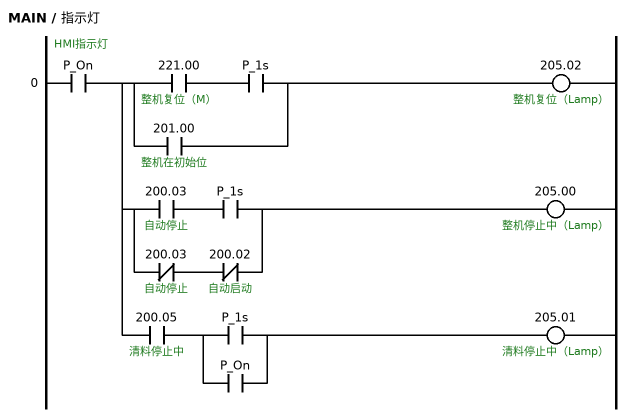
; [picture p336: MAIN / 指示灯, rungs 0-0]
; rung 0: HMI指示灯
LD P_On
OUT TR0
LD 221.00  ; 整机复位（M）
AND P_1s
OR 201.00  ; 整机在初始位
ANDLD
OUT 205.02  ; 整机复位（Lamp）
LD TR0
LD 200.03  ; 自动停止
AND P_1s
LDNOT 200.03  ; 自动停止
ANDNOT 200.02  ; 自动启动
ORLD
ANDLD
OUT 205.00  ; 整机停止中（Lamp）
LD TR0
AND 200.05  ; 清料停止中
LD P_1s
OR P_On
ANDLD
OUT 205.01  ; 清料停止中（Lamp）

### Section 外部输出

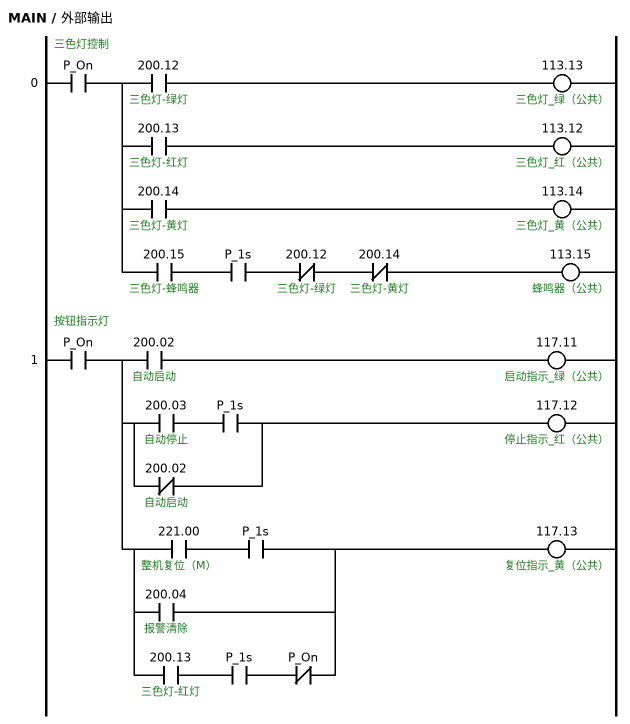
; rung 0: 三色灯控制
LD P_On
OUT TR0
AND 200.12  ; 三色灯-绿灯
OUT 113.13  ; 三色灯_绿（公共）
LD TR0
AND 200.13  ; 三色灯-红灯
OUT 113.12  ; 三色灯_红（公共）
LD TR0
AND 200.14  ; 三色灯-黄灯
OUT 113.14  ; 三色灯_黄（公共）
LD TR0
AND 200.15  ; 三色灯-蜂鸣器
AND P_1s
ANDNOT 200.12  ; 三色灯-绿灯
ANDNOT 200.14  ; 三色灯-黄灯
OUT 113.15  ; 蜂鸣器（公共）
; rung 1: 按钮指示灯
LD P_On
OUT TR0
AND 200.02  ; 自动启动
OUT 117.11  ; 启动指示_绿（公共）
LD TR0
LD 200.03  ; 自动停止
AND P_1s
ORNOT 200.02  ; 自动启动
ANDLD
OUT 117.12  ; 停止指示_红（公共）
LD TR0
LD 221.00  ; 整机复位（M）
AND P_1s
OR 200.04  ; 报警清除
LD 200.13  ; 三色灯-红灯
AND P_1s
ANDNOT P_On
ORLD
ANDLD
OUT 117.13  ; 复位指示_黄（公共）

### Section END
; rung 0
END(001)

## Program 电芯来料_RK_01 (cyclic task 1)

### Section Main

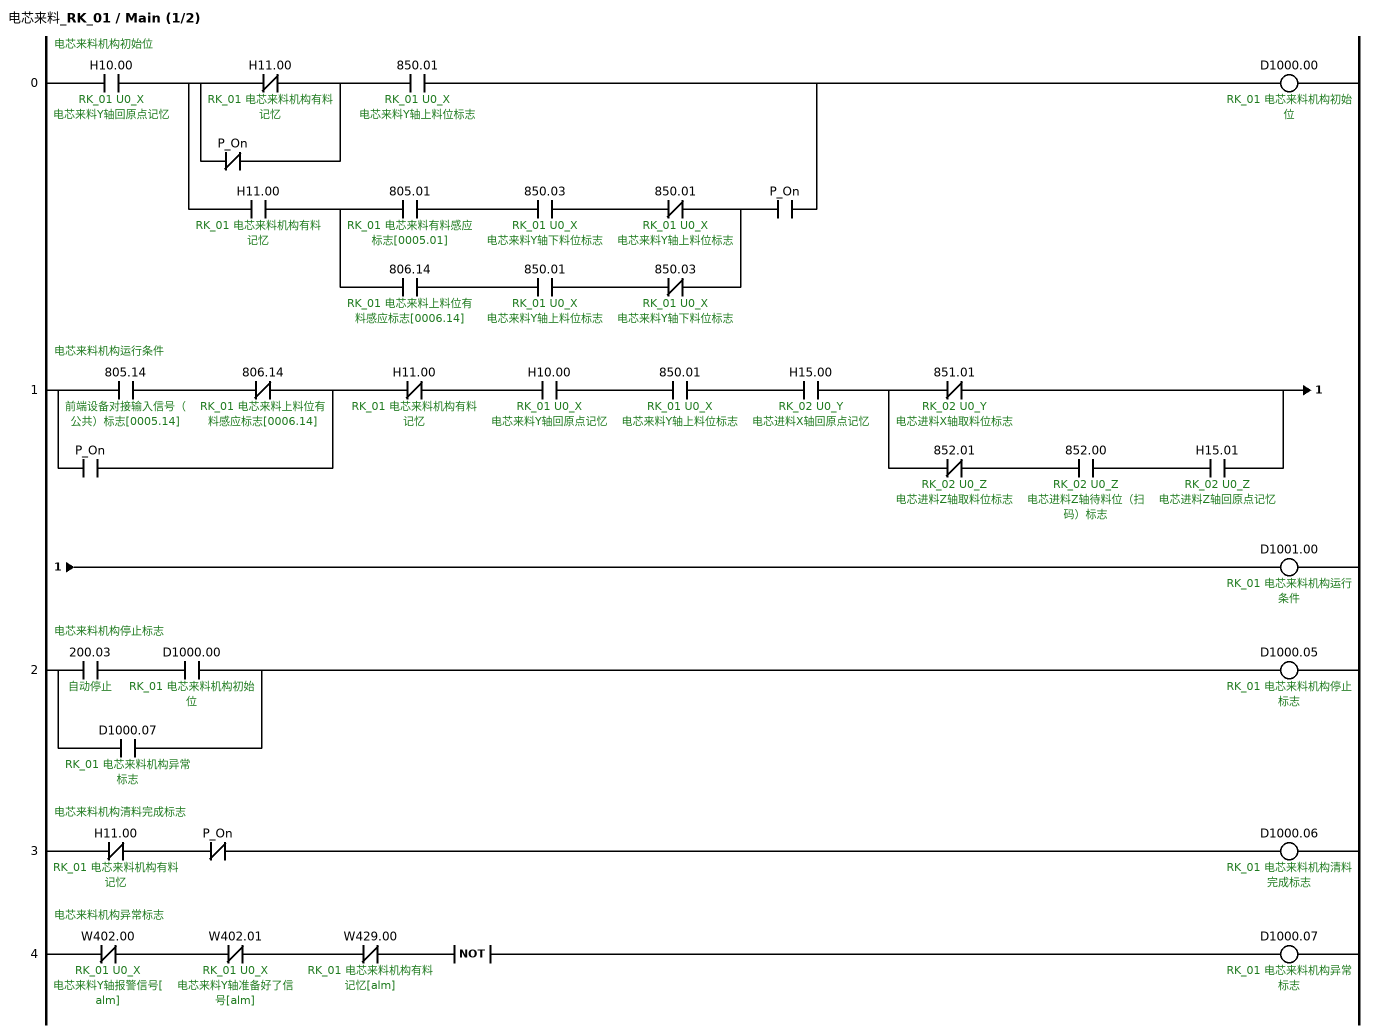
; rung 0: 电芯来料机构初始位
LD H10.00  ; RK_01 U0_X 电芯来料Y轴回原点记忆
LDNOT H11.00  ; RK_01 电芯来料机构有料记忆
ORNOT P_On
AND 850.01  ; RK_01 U0_X 电芯来料Y轴上料位标志
LD H11.00  ; RK_01 电芯来料机构有料记忆
LD 805.01  ; RK_01 电芯来料有料感应标志[0005.01]
AND 850.03  ; RK_01 U0_X 电芯来料Y轴下料位标志
ANDNOT 850.01  ; RK_01 U0_X 电芯来料Y轴上料位标志
LD 806.14  ; RK_01 电芯来料上料位有料感应标志[0006.14]
AND 850.01  ; RK_01 U0_X 电芯来料Y轴上料位标志
ANDNOT 850.03  ; RK_01 U0_X 电芯来料Y轴下料位标志
ORLD
ANDLD
AND P_On
ORLD
ANDLD
OUT D1000.00  ; RK_01 电芯来料机构初始位
; rung 1: 电芯来料机构运行条件
LD 805.14  ; 前端设备对接输入信号（公共）标志[0005.14]  // 前端设备放料中（放料中=1）！
ANDNOT 806.14  ; RK_01 电芯来料上料位有料感应标志[0006.14]
OR P_On
ANDNOT H11.00  ; RK_01 电芯来料机构有料记忆
AND H10.00  ; RK_01 U0_X 电芯来料Y轴回原点记忆
AND 850.01  ; RK_01 U0_X 电芯来料Y轴上料位标志
AND H15.00  ; RK_02 U0_Y 电芯进料X轴回原点记忆
LDNOT 851.01  ; RK_02 U0_Y 电芯进料X轴取料位标志
LDNOT 852.01  ; RK_02 U0_Z 电芯进料Z轴取料位标志
AND 852.00  ; RK_02 U0_Z 电芯进料Z轴待料位（扫码）标志
AND H15.01  ; RK_02 U0_Z 电芯进料Z轴回原点记忆
ORLD
ANDLD
OUT D1001.00  ; RK_01 电芯来料机构运行条件
; rung 2: 电芯来料机构停止标志
LD 200.03  ; 自动停止
AND D1000.00  ; RK_01 电芯来料机构初始位
OR D1000.07  ; RK_01 电芯来料机构异常标志
OUT D1000.05  ; RK_01 电芯来料机构停止标志
; rung 3: 电芯来料机构清料完成标志
LDNOT H11.00  ; RK_01 电芯来料机构有料记忆
ANDNOT P_On  // 上料位非扫码完成料，清料时无需考虑！！
OUT D1000.06  ; RK_01 电芯来料机构清料完成标志
; rung 4: 电芯来料机构异常标志
LDNOT W402.00  ; RK_01 U0_X 电芯来料Y轴报警信号[alm]
ANDNOT W402.01  ; RK_01 U0_X 电芯来料Y轴准备好了信号[alm]
ANDNOT W429.00  ; RK_01 电芯来料机构有料记忆[alm]
NOT(520)
OUT D1000.07  ; RK_01 电芯来料机构异常标志

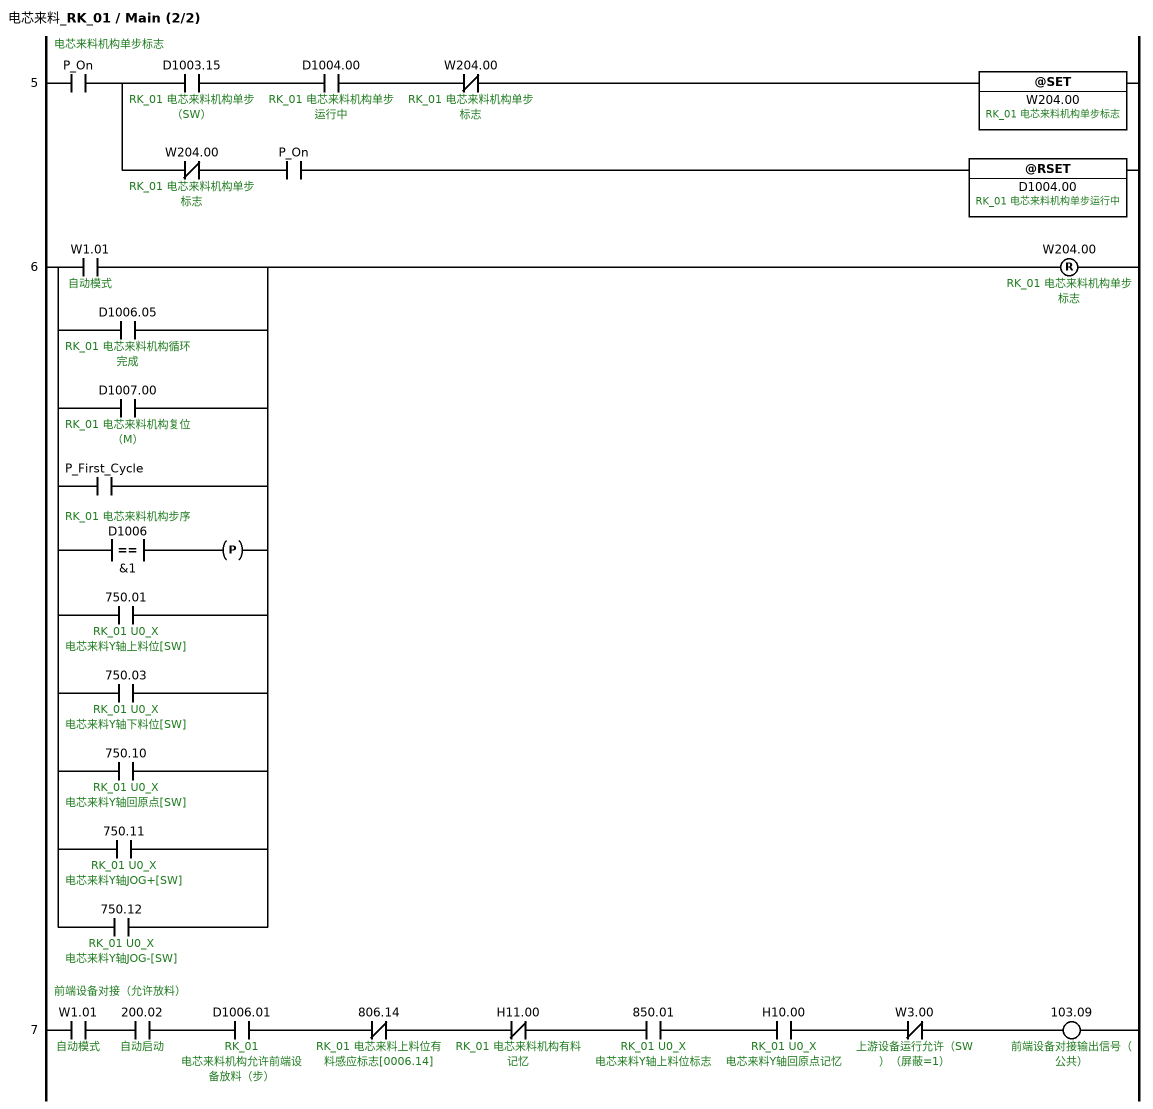
; rung 5: 电芯来料机构单步标志
LD P_On
OUT TR0
AND D1003.15  ; RK_01 电芯来料机构单步（SW）
AND D1004.00  ; RK_01 电芯来料机构单步运行中
ANDNOT W204.00  ; RK_01 电芯来料机构单步标志
@SET W204.00  ; RK_01 电芯来料机构单步标志
LD TR0
ANDNOT W204.00  ; RK_01 电芯来料机构单步标志
AND P_On
@RSET D1004.00  ; RK_01 电芯来料机构单步运行中
; rung 6
LD W1.01  ; 自动模式
OR D1006.05  ; RK_01 电芯来料机构循环完成
OR D1007.00  ; RK_01 电芯来料机构复位（M）
OR P_First_Cycle
LD=(300) D1006 &1  ; RK_01 电芯来料机构步序
UP(521)
ORLD
OR 750.01  ; RK_01 U0_X 电芯来料Y轴上料位[SW]
OR 750.03  ; RK_01 U0_X 电芯来料Y轴下料位[SW]
OR 750.10  ; RK_01 U0_X 电芯来料Y轴回原点[SW]
OR 750.11  ; RK_01 U0_X 电芯来料Y轴JOG+[SW]
OR 750.12  ; RK_01 U0_X 电芯来料Y轴JOG-[SW]
RSET W204.00  ; RK_01 电芯来料机构单步标志
; rung 7: 前端设备对接（允许放料）
LD W1.01  ; 自动模式
AND 200.02  ; 自动启动
AND D1006.01  ; RK_01  电芯来料机构允许前端设备放料（步）
ANDNOT 806.14  ; RK_01 电芯来料上料位有料感应标志[0006.14]
ANDNOT H11.00  ; RK_01 电芯来料机构有料记忆
AND 850.01  ; RK_01 U0_X 电芯来料Y轴上料位标志
AND H10.00  ; RK_01 U0_X 电芯来料Y轴回原点记忆
ANDNOT W3.00  ; 上游设备运行允许（SW）（屏蔽=1）
OUT 103.09  ; 前端设备对接输出信号（公共）

### Section 手动

### Section 自动

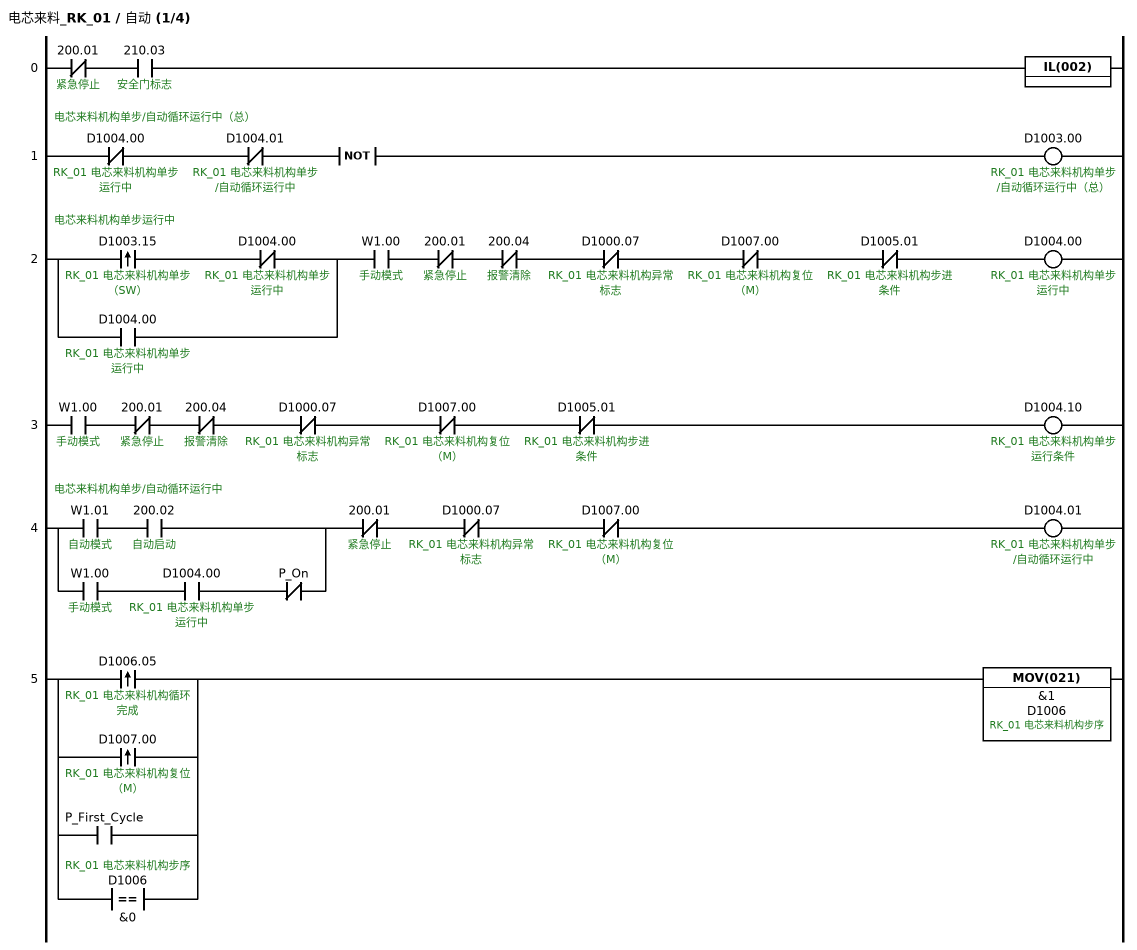
; rung 0
LDNOT 200.01  ; 紧急停止
AND 210.03  ; 安全门标志
IL(002)
; rung 1: 电芯来料机构单步/自动循环运行中（总）
LDNOT D1004.00  ; RK_01 电芯来料机构单步运行中
ANDNOT D1004.01  ; RK_01 电芯来料机构单步/自动循环运行中
NOT(520)
OUT D1003.00  ; RK_01 电芯来料机构单步/自动循环运行中（总）
; rung 2: 电芯来料机构单步运行中
@LD D1003.15  ; RK_01 电芯来料机构单步（SW）
ANDNOT D1004.00  ; RK_01 电芯来料机构单步运行中
OR D1004.00  ; RK_01 电芯来料机构单步运行中
AND W1.00  ; 手动模式
ANDNOT 200.01  ; 紧急停止
ANDNOT 200.04  ; 报警清除
ANDNOT D1000.07  ; RK_01 电芯来料机构异常标志
ANDNOT D1007.00  ; RK_01 电芯来料机构复位（M）
ANDNOT D1005.01  ; RK_01 电芯来料机构步进条件
OUT D1004.00  ; RK_01 电芯来料机构单步运行中
; rung 3
LD W1.00  ; 手动模式
ANDNOT 200.01  ; 紧急停止
ANDNOT 200.04  ; 报警清除
ANDNOT D1000.07  ; RK_01 电芯来料机构异常标志
ANDNOT D1007.00  ; RK_01 电芯来料机构复位（M）
ANDNOT D1005.01  ; RK_01 电芯来料机构步进条件
OUT D1004.10  ; RK_01 电芯来料机构单步运行条件
; rung 4: 电芯来料机构单步/自动循环运行中
LD W1.01  ; 自动模式
AND 200.02  ; 自动启动
LD W1.00  ; 手动模式
AND D1004.00  ; RK_01 电芯来料机构单步运行中
ANDNOT P_On
ORLD
ANDNOT 200.01  ; 紧急停止
ANDNOT D1000.07  ; RK_01 电芯来料机构异常标志
ANDNOT D1007.00  ; RK_01 电芯来料机构复位（M）
OUT D1004.01  ; RK_01 电芯来料机构单步/自动循环运行中
; rung 5
@LD D1006.05  ; RK_01 电芯来料机构循环完成
@OR D1007.00  ; RK_01 电芯来料机构复位（M）
OR P_First_Cycle
OR=(300) D1006 &0  ; RK_01 电芯来料机构步序
MOV(021) &1 D1006  ; RK_01 电芯来料机构步序

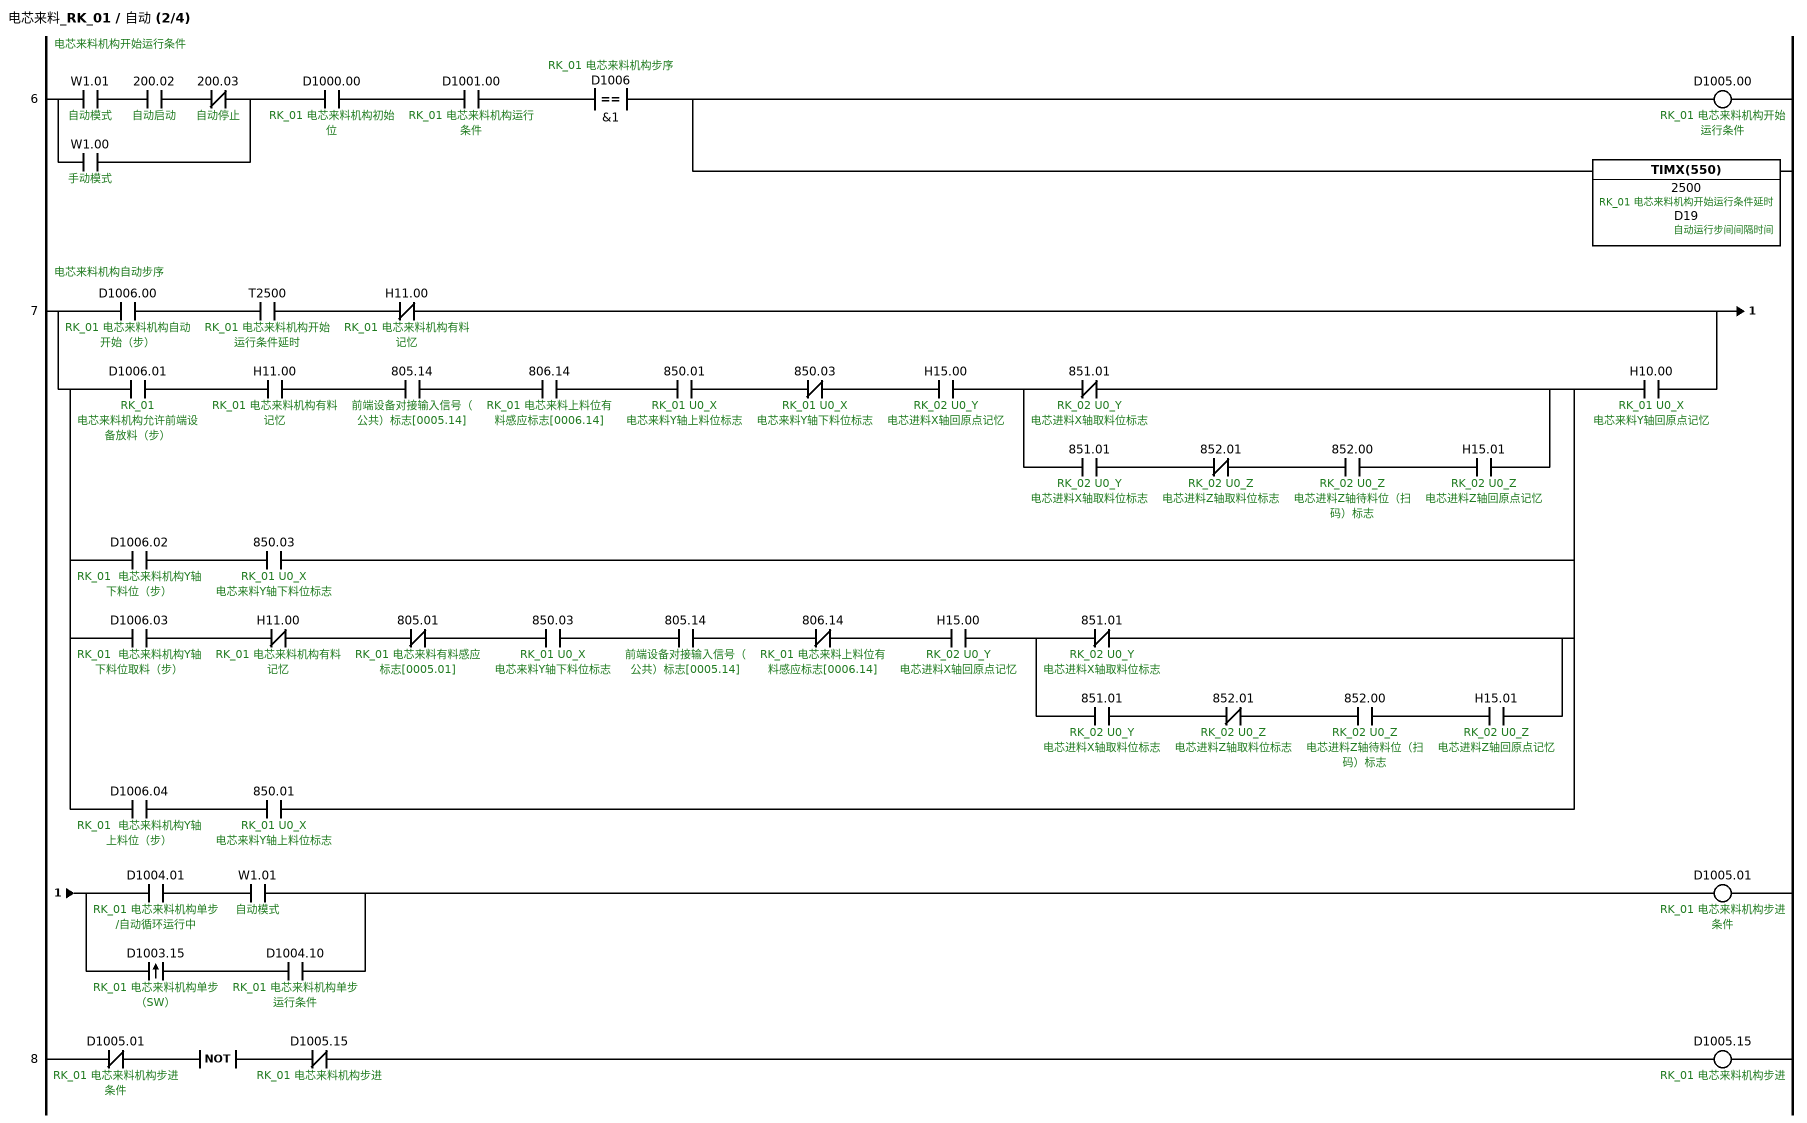
; rung 6: 电芯来料机构开始运行条件
LD W1.01  ; 自动模式
AND 200.02  ; 自动启动
ANDNOT 200.03  ; 自动停止
OR W1.00  ; 手动模式
AND D1000.00  ; RK_01 电芯来料机构初始位
AND D1001.00  ; RK_01 电芯来料机构运行条件
AND=(300) D1006 &1  ; RK_01 电芯来料机构步序
OUT D1005.00  ; RK_01 电芯来料机构开始运行条件
TIMX(550) 2500 D19  ; 自动运行步间间隔时间, RK_01 电芯来料机构开始运行条件延时
; rung 7: 电芯来料机构自动步序
LD D1006.00  ; RK_01 电芯来料机构自动开始（步）
AND T2500  ; RK_01 电芯来料机构开始运行条件延时
ANDNOT H11.00  ; RK_01 电芯来料机构有料记忆
LD D1006.01  ; RK_01  电芯来料机构允许前端设备放料（步）
AND H11.00  ; RK_01 电芯来料机构有料记忆
AND 805.14  ; 前端设备对接输入信号（公共）标志[0005.14]  // 前端设备放料中（放料中=1）！
AND 806.14  ; RK_01 电芯来料上料位有料感应标志[0006.14]
AND 850.01  ; RK_01 U0_X 电芯来料Y轴上料位标志
ANDNOT 850.03  ; RK_01 U0_X 电芯来料Y轴下料位标志
AND H15.00  ; RK_02 U0_Y 电芯进料X轴回原点记忆
LDNOT 851.01  ; RK_02 U0_Y 电芯进料X轴取料位标志
LD 851.01  ; RK_02 U0_Y 电芯进料X轴取料位标志
ANDNOT 852.01  ; RK_02 U0_Z 电芯进料Z轴取料位标志
AND 852.00  ; RK_02 U0_Z 电芯进料Z轴待料位（扫码）标志
AND H15.01  ; RK_02 U0_Z 电芯进料Z轴回原点记忆
ORLD
ANDLD
LD D1006.02  ; RK_01  电芯来料机构Y轴下料位（步）
AND 850.03  ; RK_01 U0_X 电芯来料Y轴下料位标志
ORLD
LD D1006.03  ; RK_01  电芯来料机构Y轴下料位取料（步）
ANDNOT H11.00  ; RK_01 电芯来料机构有料记忆
ANDNOT 805.01  ; RK_01 电芯来料有料感应标志[0005.01]
AND 850.03  ; RK_01 U0_X 电芯来料Y轴下料位标志
AND 805.14  ; 前端设备对接输入信号（公共）标志[0005.14]  // 前端设备放料中（放料中=1）！
ANDNOT 806.14  ; RK_01 电芯来料上料位有料感应标志[0006.14]
AND H15.00  ; RK_02 U0_Y 电芯进料X轴回原点记忆
LDNOT 851.01  ; RK_02 U0_Y 电芯进料X轴取料位标志
LD 851.01  ; RK_02 U0_Y 电芯进料X轴取料位标志
ANDNOT 852.01  ; RK_02 U0_Z 电芯进料Z轴取料位标志
AND 852.00  ; RK_02 U0_Z 电芯进料Z轴待料位（扫码）标志
AND H15.01  ; RK_02 U0_Z 电芯进料Z轴回原点记忆
ORLD
ANDLD
ORLD
LD D1006.04  ; RK_01  电芯来料机构Y轴上料位（步）
AND 850.01  ; RK_01 U0_X 电芯来料Y轴上料位标志
ORLD
AND H10.00  ; RK_01 U0_X 电芯来料Y轴回原点记忆
ORLD
LD D1004.01  ; RK_01 电芯来料机构单步/自动循环运行中
AND W1.01  ; 自动模式
@LD D1003.15  ; RK_01 电芯来料机构单步（SW）
AND D1004.10  ; RK_01 电芯来料机构单步运行条件
ORLD
ANDLD
OUT D1005.01  ; RK_01 电芯来料机构步进条件
; rung 8
LDNOT D1005.01  ; RK_01 电芯来料机构步进条件
NOT(520)
ANDNOT D1005.15  ; RK_01 电芯来料机构步进
OUT D1005.15  ; RK_01 电芯来料机构步进

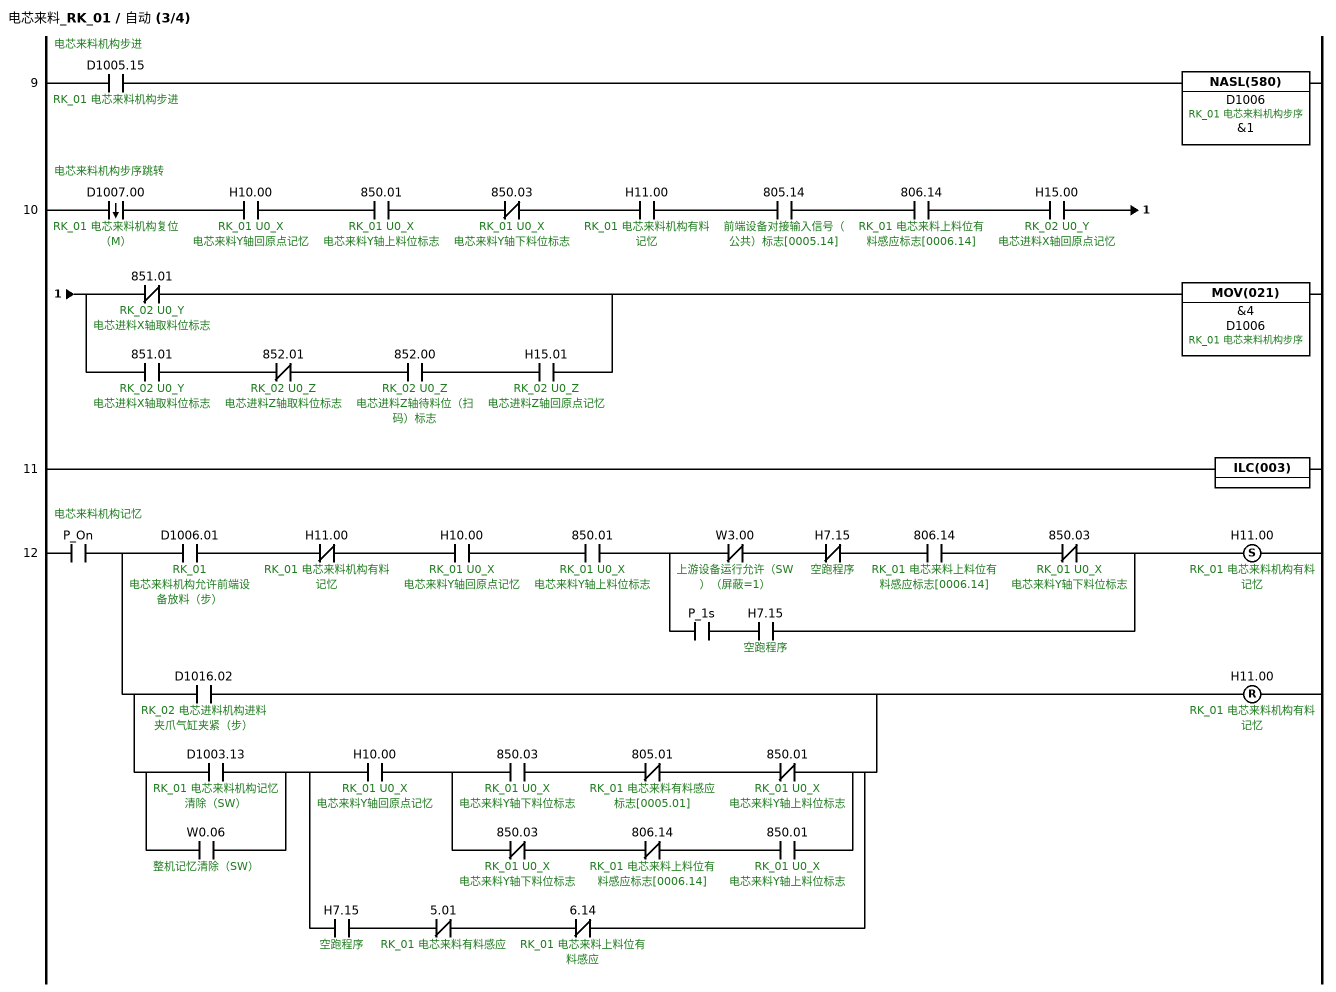
; rung 9: 电芯来料机构步进
LD D1005.15  ; RK_01 电芯来料机构步进
NASL(580) D1006 &1  ; RK_01 电芯来料机构步序
; rung 10: 电芯来料机构步序跳转
%LD D1007.00  ; RK_01 电芯来料机构复位（M）
AND H10.00  ; RK_01 U0_X 电芯来料Y轴回原点记忆
AND 850.01  ; RK_01 U0_X 电芯来料Y轴上料位标志
ANDNOT 850.03  ; RK_01 U0_X 电芯来料Y轴下料位标志
AND H11.00  ; RK_01 电芯来料机构有料记忆
AND 805.14  ; 前端设备对接输入信号（公共）标志[0005.14]  // 前端设备放料中（放料中=1）！
AND 806.14  ; RK_01 电芯来料上料位有料感应标志[0006.14]
AND H15.00  ; RK_02 U0_Y 电芯进料X轴回原点记忆
LDNOT 851.01  ; RK_02 U0_Y 电芯进料X轴取料位标志
LD 851.01  ; RK_02 U0_Y 电芯进料X轴取料位标志
ANDNOT 852.01  ; RK_02 U0_Z 电芯进料Z轴取料位标志
AND 852.00  ; RK_02 U0_Z 电芯进料Z轴待料位（扫码）标志
AND H15.01  ; RK_02 U0_Z 电芯进料Z轴回原点记忆
ORLD
ANDLD
MOV(021) &4 D1006  ; RK_01 电芯来料机构步序  // RK_01  电芯来料机构Y轴下料位步（D1006.02）
; rung 11
ILC(003)
; rung 12: 电芯来料机构记忆
LD P_On
OUT TR0
AND D1006.01  ; RK_01  电芯来料机构允许前端设备放料（步）
ANDNOT H11.00  ; RK_01 电芯来料机构有料记忆
AND H10.00  ; RK_01 U0_X 电芯来料Y轴回原点记忆
AND 850.01  ; RK_01 U0_X 电芯来料Y轴上料位标志
LDNOT W3.00  ; 上游设备运行允许（SW）（屏蔽=1）
ANDNOT H7.15  ; 空跑程序
AND 806.14  ; RK_01 电芯来料上料位有料感应标志[0006.14]
ANDNOT 850.03  ; RK_01 U0_X 电芯来料Y轴下料位标志
LD P_1s
AND H7.15  ; 空跑程序
ORLD
ANDLD
SET H11.00  ; RK_01 电芯来料机构有料记忆
LD TR0
LD D1016.02  ; RK_02 电芯进料机构进料夹爪气缸夹紧（步）
LD D1003.13  ; RK_01 电芯来料机构记忆清除（SW）
OR W0.06  ; 整机记忆清除（SW）
LD H10.00  ; RK_01 U0_X 电芯来料Y轴回原点记忆
LD 850.03  ; RK_01 U0_X 电芯来料Y轴下料位标志
ANDNOT 805.01  ; RK_01 电芯来料有料感应标志[0005.01]
ANDNOT 850.01  ; RK_01 U0_X 电芯来料Y轴上料位标志
LDNOT 850.03  ; RK_01 U0_X 电芯来料Y轴下料位标志
ANDNOT 806.14  ; RK_01 电芯来料上料位有料感应标志[0006.14]
AND 850.01  ; RK_01 U0_X 电芯来料Y轴上料位标志
ORLD
ANDLD
LD H7.15  ; 空跑程序
ANDNOT 5.01  ; RK_01 电芯来料有料感应
ANDNOT 6.14  ; RK_01 电芯来料上料位有料感应
ORLD
ANDLD
ORLD
ANDLD
RSET H11.00  ; RK_01 电芯来料机构有料记忆

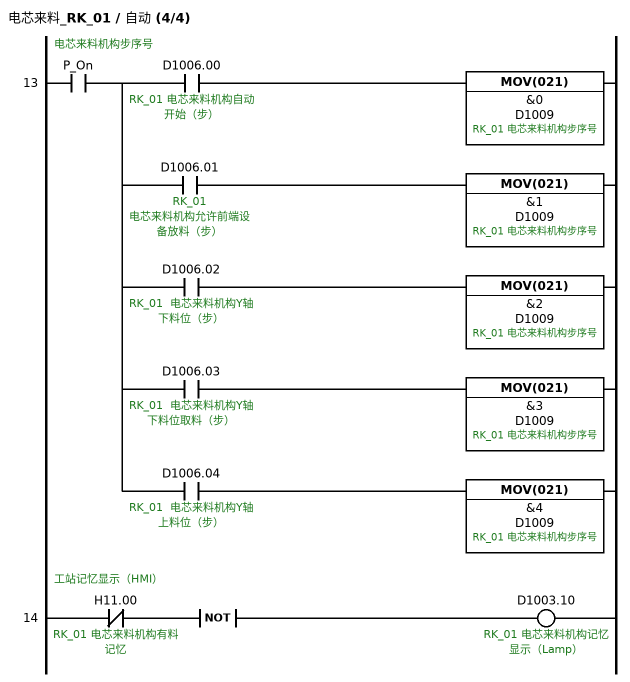
; rung 13: 电芯来料机构步序号
LD P_On
OUT TR0
AND D1006.00  ; RK_01 电芯来料机构自动开始（步）
MOV(021) &0 D1009  ; RK_01 电芯来料机构步序号
LD TR0
AND D1006.01  ; RK_01  电芯来料机构允许前端设备放料（步）
MOV(021) &1 D1009  ; RK_01 电芯来料机构步序号
LD TR0
AND D1006.02  ; RK_01  电芯来料机构Y轴下料位（步）
MOV(021) &2 D1009  ; RK_01 电芯来料机构步序号
LD TR0
AND D1006.03  ; RK_01  电芯来料机构Y轴下料位取料（步）
MOV(021) &3 D1009  ; RK_01 电芯来料机构步序号
LD TR0
AND D1006.04  ; RK_01  电芯来料机构Y轴上料位（步）
MOV(021) &4 D1009  ; RK_01 电芯来料机构步序号
; rung 14: 工站记忆显示（HMI）
LDNOT H11.00  ; RK_01 电芯来料机构有料记忆
NOT(520)
OUT D1003.10  ; RK_01 电芯来料机构记忆显示（Lamp）

### Section 复位

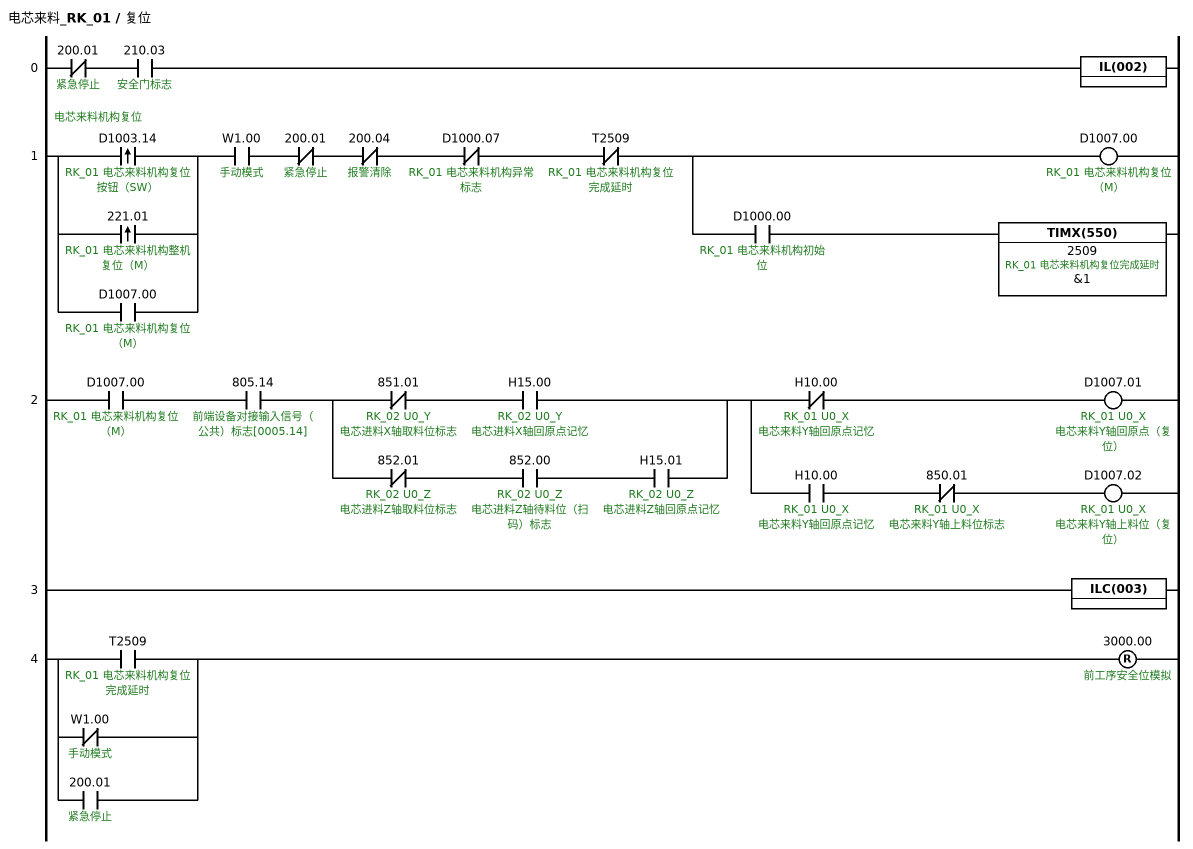
; rung 0
LDNOT 200.01  ; 紧急停止
AND 210.03  ; 安全门标志
IL(002)
; rung 1: 电芯来料机构复位
@LD D1003.14  ; RK_01 电芯来料机构复位按钮（SW）
@OR 221.01  ; RK_01 电芯来料机构整机复位（M）
OR D1007.00  ; RK_01 电芯来料机构复位（M）
AND W1.00  ; 手动模式
ANDNOT 200.01  ; 紧急停止
ANDNOT 200.04  ; 报警清除
ANDNOT D1000.07  ; RK_01 电芯来料机构异常标志
ANDNOT T2509  ; RK_01 电芯来料机构复位完成延时
OUT D1007.00  ; RK_01 电芯来料机构复位（M）
AND D1000.00  ; RK_01 电芯来料机构初始位
TIMX(550) 2509 &1  ; RK_01 电芯来料机构复位完成延时
; rung 2
LD D1007.00  ; RK_01 电芯来料机构复位（M）
AND 805.14  ; 前端设备对接输入信号（公共）标志[0005.14]  // 前端设备放料中（放料中=1）！
LDNOT 851.01  ; RK_02 U0_Y 电芯进料X轴取料位标志
AND H15.00  ; RK_02 U0_Y 电芯进料X轴回原点记忆
LDNOT 852.01  ; RK_02 U0_Z 电芯进料Z轴取料位标志
AND 852.00  ; RK_02 U0_Z 电芯进料Z轴待料位（扫码）标志
AND H15.01  ; RK_02 U0_Z 电芯进料Z轴回原点记忆
ORLD
ANDLD
OUT TR0
ANDNOT H10.00  ; RK_01 U0_X 电芯来料Y轴回原点记忆
OUT D1007.01  ; RK_01 U0_X 电芯来料Y轴回原点（复位）
LD TR0
AND H10.00  ; RK_01 U0_X 电芯来料Y轴回原点记忆
ANDNOT 850.01  ; RK_01 U0_X 电芯来料Y轴上料位标志
OUT D1007.02  ; RK_01 U0_X 电芯来料Y轴上料位（复位）
; rung 3
ILC(003)
; rung 4
LD T2509  ; RK_01 电芯来料机构复位完成延时
ORNOT W1.00  ; 手动模式
OR 200.01  ; 紧急停止
RSET 3000.00  ; 前工序安全位模拟

### Section 指示灯

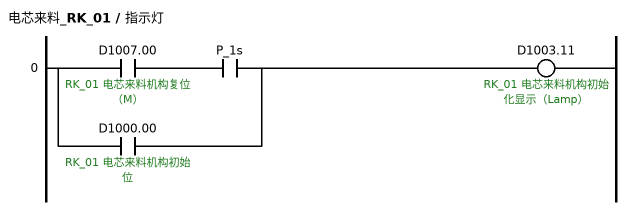
; rung 0
LD D1007.00  ; RK_01 电芯来料机构复位（M）
AND P_1s
OR D1000.00  ; RK_01 电芯来料机构初始位
OUT D1003.11  ; RK_01 电芯来料机构初始化显示（Lamp）

### Section 外部输出

### Section END
; rung 0
END(001)

## Program 电芯进料_RK_02 (cyclic task 2)
Local symbols
NOT BOOL

### Section Main

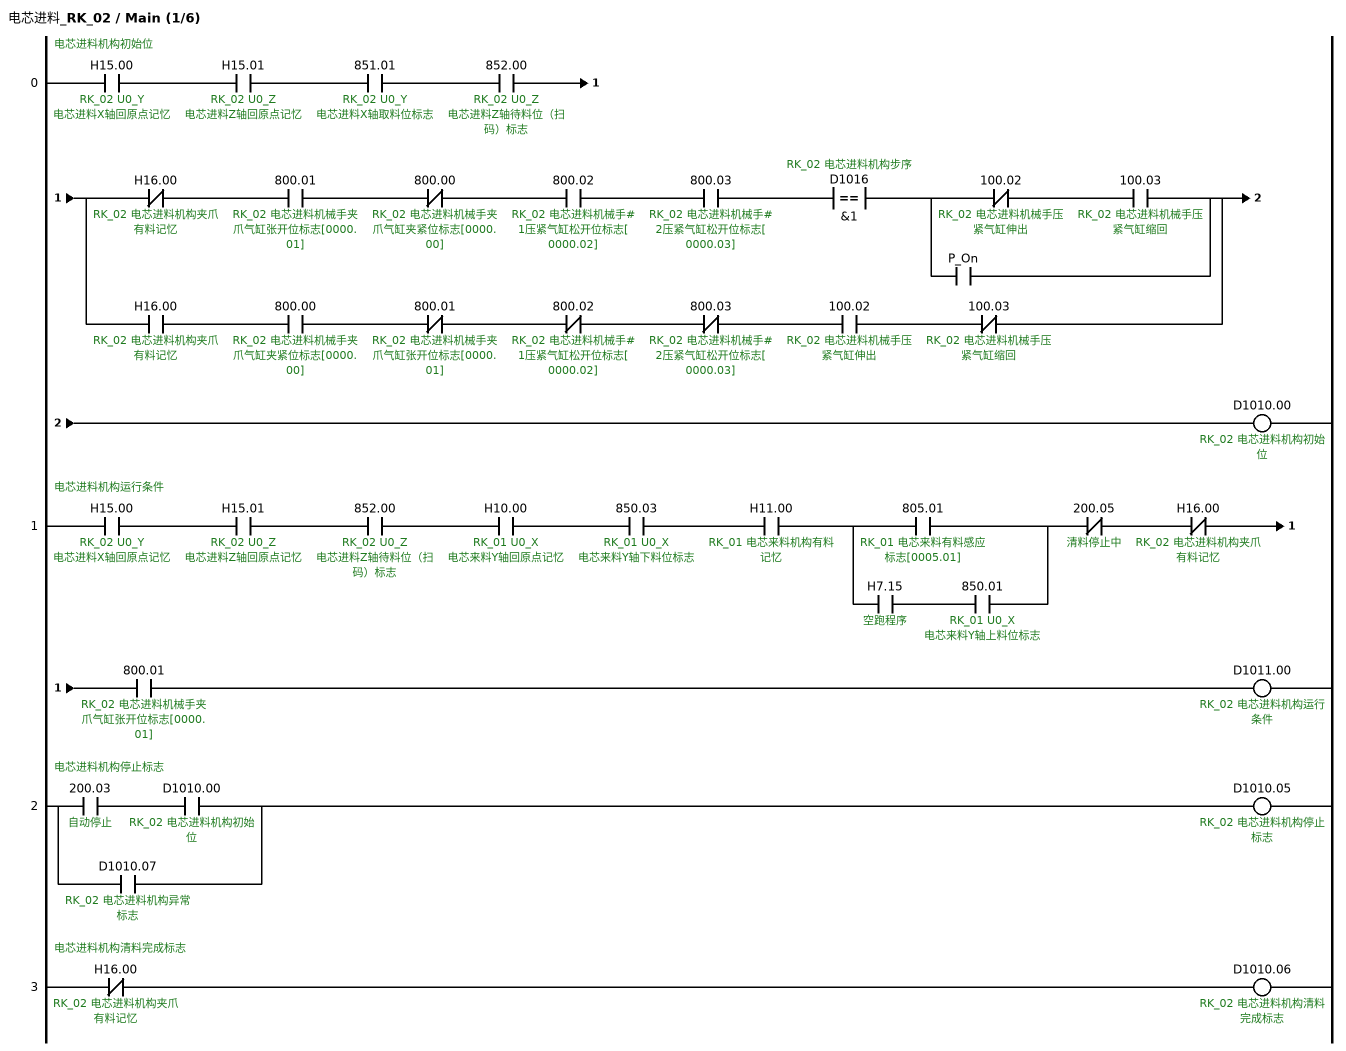
; rung 0: 电芯进料机构初始位
LD H15.00  ; RK_02 U0_Y 电芯进料X轴回原点记忆
AND H15.01  ; RK_02 U0_Z 电芯进料Z轴回原点记忆
AND 851.01  ; RK_02 U0_Y 电芯进料X轴取料位标志
AND 852.00  ; RK_02 U0_Z 电芯进料Z轴待料位（扫码）标志
LDNOT H16.00  ; RK_02 电芯进料机构夹爪有料记忆
AND 800.01  ; RK_02 电芯进料机械手夹爪气缸张开位标志[0000.01]
ANDNOT 800.00  ; RK_02 电芯进料机械手夹爪气缸夹紧位标志[0000.00]
AND 800.02  ; RK_02 电芯进料机械手#1压紧气缸松开位标志[0000.02]
AND 800.03  ; RK_02 电芯进料机械手#2压紧气缸松开位标志[0000.03]
AND=(300) D1016 &1  ; RK_02 电芯进料机构步序
LDNOT 100.02  ; RK_02 电芯进料机械手压紧气缸伸出
AND 100.03  ; RK_02 电芯进料机械手压紧气缸缩回
OR P_On
ANDLD
LD H16.00  ; RK_02 电芯进料机构夹爪有料记忆
AND 800.00  ; RK_02 电芯进料机械手夹爪气缸夹紧位标志[0000.00]
ANDNOT 800.01  ; RK_02 电芯进料机械手夹爪气缸张开位标志[0000.01]
ANDNOT 800.02  ; RK_02 电芯进料机械手#1压紧气缸松开位标志[0000.02]
ANDNOT 800.03  ; RK_02 电芯进料机械手#2压紧气缸松开位标志[0000.03]
AND 100.02  ; RK_02 电芯进料机械手压紧气缸伸出
ANDNOT 100.03  ; RK_02 电芯进料机械手压紧气缸缩回
ORLD
ANDLD
OUT D1010.00  ; RK_02 电芯进料机构初始位
; rung 1: 电芯进料机构运行条件
LD H15.00  ; RK_02 U0_Y 电芯进料X轴回原点记忆
AND H15.01  ; RK_02 U0_Z 电芯进料Z轴回原点记忆
AND 852.00  ; RK_02 U0_Z 电芯进料Z轴待料位（扫码）标志
AND H10.00  ; RK_01 U0_X 电芯来料Y轴回原点记忆
AND 850.03  ; RK_01 U0_X 电芯来料Y轴下料位标志
AND H11.00  ; RK_01 电芯来料机构有料记忆
LD 805.01  ; RK_01 电芯来料有料感应标志[0005.01]
LD H7.15  ; 空跑程序
AND 850.01  ; RK_01 U0_X 电芯来料Y轴上料位标志
ORLD
ANDLD
ANDNOT 200.05  ; 清料停止中
ANDNOT H16.00  ; RK_02 电芯进料机构夹爪有料记忆
AND 800.01  ; RK_02 电芯进料机械手夹爪气缸张开位标志[0000.01]
OUT D1011.00  ; RK_02 电芯进料机构运行条件
; rung 2: 电芯进料机构停止标志
LD 200.03  ; 自动停止
AND D1010.00  ; RK_02 电芯进料机构初始位
OR D1010.07  ; RK_02 电芯进料机构异常标志
OUT D1010.05  ; RK_02 电芯进料机构停止标志
; rung 3: 电芯进料机构清料完成标志
LDNOT H16.00  ; RK_02 电芯进料机构夹爪有料记忆
OUT D1010.06  ; RK_02 电芯进料机构清料完成标志

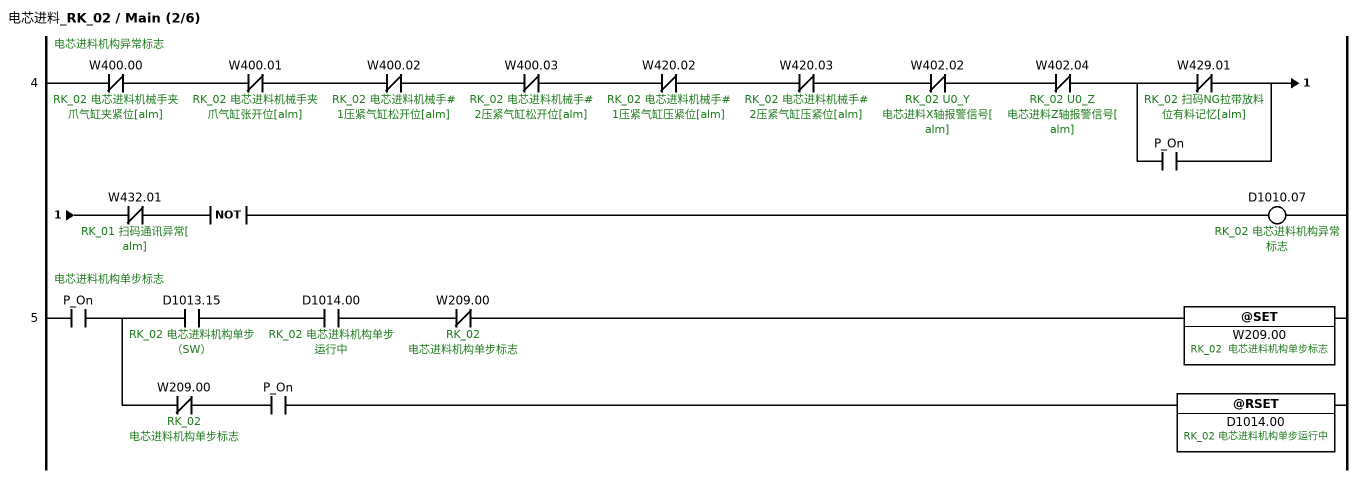
; rung 4: 电芯进料机构异常标志
LDNOT W400.00  ; RK_02 电芯进料机械手夹爪气缸夹紧位[alm]
ANDNOT W400.01  ; RK_02 电芯进料机械手夹爪气缸张开位[alm]
ANDNOT W400.02  ; RK_02 电芯进料机械手#1压紧气缸松开位[alm]
ANDNOT W400.03  ; RK_02 电芯进料机械手#2压紧气缸松开位[alm]
ANDNOT W420.02  ; RK_02 电芯进料机械手#1压紧气缸压紧位[alm]
ANDNOT W420.03  ; RK_02 电芯进料机械手#2压紧气缸压紧位[alm]
ANDNOT W402.02  ; RK_02 U0_Y 电芯进料X轴报警信号[alm]
ANDNOT W402.04  ; RK_02 U0_Z 电芯进料Z轴报警信号[alm]
LDNOT W429.01  ; RK_02 扫码NG拉带放料位有料记忆[alm]
OR P_On
ANDLD
ANDNOT W432.01  ; RK_01 扫码通讯异常[alm]
NOT(520)
OUT D1010.07  ; RK_02 电芯进料机构异常标志
; rung 5: 电芯进料机构单步标志
LD P_On
OUT TR0
AND D1013.15  ; RK_02 电芯进料机构单步（SW）
AND D1014.00  ; RK_02 电芯进料机构单步运行中
ANDNOT W209.00  ; RK_02  电芯进料机构单步标志
@SET W209.00  ; RK_02  电芯进料机构单步标志
LD TR0
ANDNOT W209.00  ; RK_02  电芯进料机构单步标志
AND P_On
@RSET D1014.00  ; RK_02 电芯进料机构单步运行中

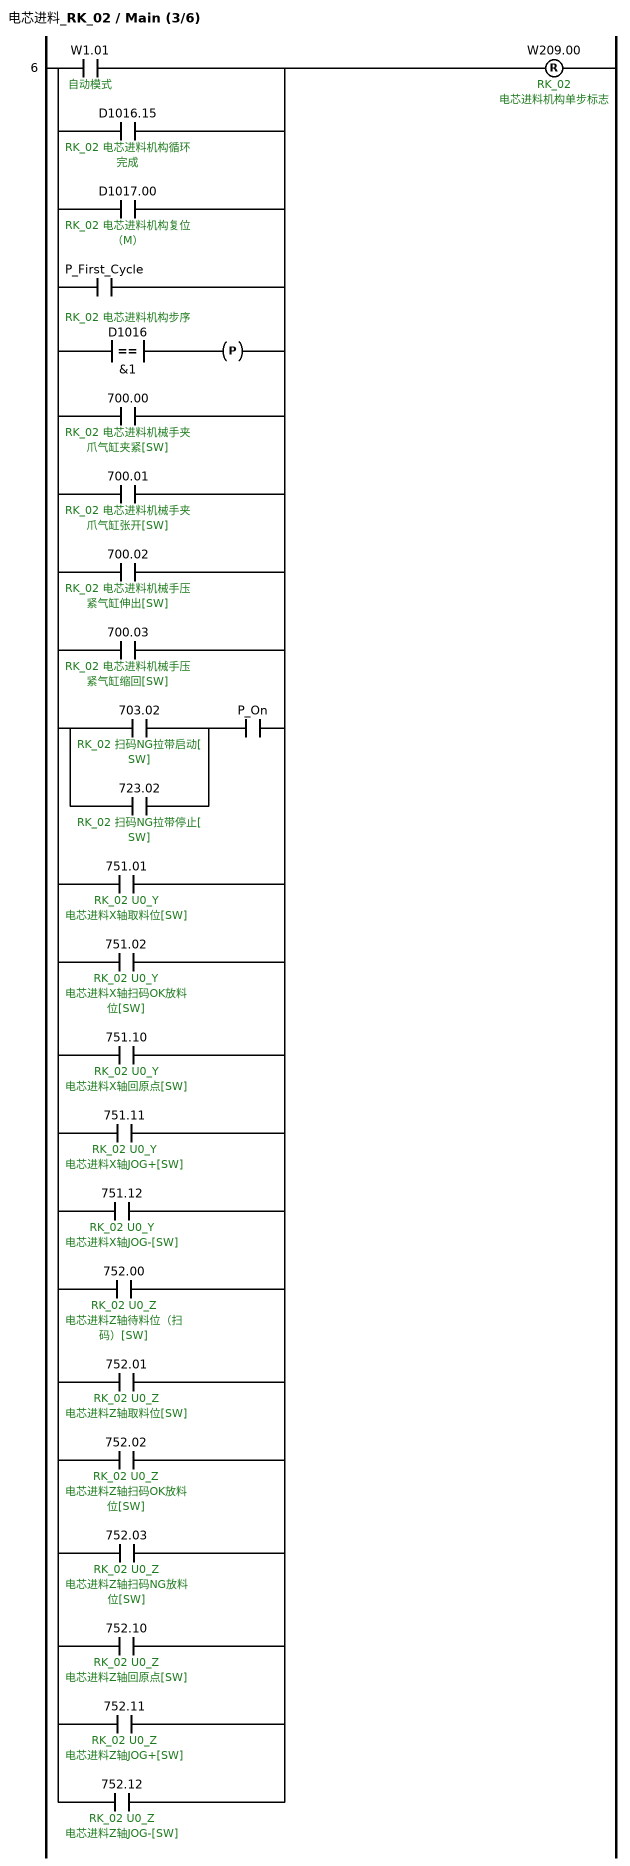
; rung 6
LD W1.01  ; 自动模式
OR D1016.15  ; RK_02 电芯进料机构循环完成
OR D1017.00  ; RK_02 电芯进料机构复位（M）
OR P_First_Cycle
LD=(300) D1016 &1  ; RK_02 电芯进料机构步序
UP(521)
ORLD
OR 700.00  ; RK_02 电芯进料机械手夹爪气缸夹紧[SW]
OR 700.01  ; RK_02 电芯进料机械手夹爪气缸张开[SW]
OR 700.02  ; RK_02 电芯进料机械手压紧气缸伸出[SW]
OR 700.03  ; RK_02 电芯进料机械手压紧气缸缩回[SW]
LD 703.02  ; RK_02 扫码NG拉带启动[SW]
OR 723.02  ; RK_02 扫码NG拉带停止[SW]
AND P_On
ORLD
OR 751.01  ; RK_02 U0_Y 电芯进料X轴取料位[SW]
OR 751.02  ; RK_02 U0_Y 电芯进料X轴扫码OK放料位[SW]
OR 751.10  ; RK_02 U0_Y 电芯进料X轴回原点[SW]
OR 751.11  ; RK_02 U0_Y 电芯进料X轴JOG+[SW]
OR 751.12  ; RK_02 U0_Y 电芯进料X轴JOG-[SW]
OR 752.00  ; RK_02 U0_Z 电芯进料Z轴待料位（扫码）[SW]
OR 752.01  ; RK_02 U0_Z 电芯进料Z轴取料位[SW]
OR 752.02  ; RK_02 U0_Z 电芯进料Z轴扫码OK放料位[SW]
OR 752.03  ; RK_02 U0_Z 电芯进料Z轴扫码NG放料位[SW]
OR 752.10  ; RK_02 U0_Z 电芯进料Z轴回原点[SW]
OR 752.11  ; RK_02 U0_Z 电芯进料Z轴JOG+[SW]
OR 752.12  ; RK_02 U0_Z 电芯进料Z轴JOG-[SW]
RSET W209.00  ; RK_02  电芯进料机构单步标志

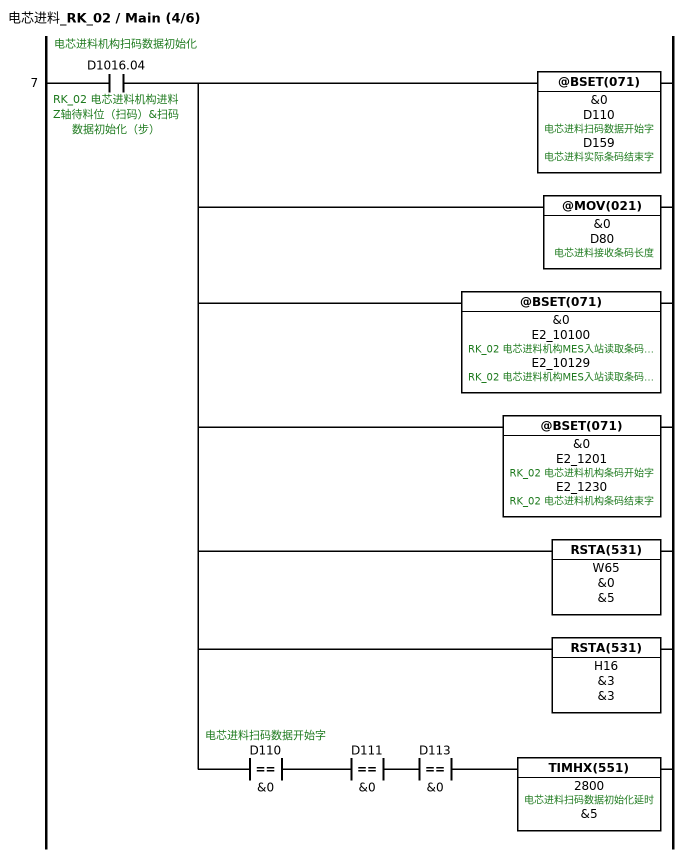
; rung 7: 电芯进料机构扫码数据初始化
LD D1016.04  ; RK_02 电芯进料机构进料Z轴待料位（扫码）&扫码数据初始化（步）
@BSET(071) &0 D110 D159  ; 电芯进料扫码数据开始字, 电芯进料实际条码结束字
@MOV(021) &0 D80  ; 电芯进料接收条码长度
@BSET(071) &0 E2_10100 E2_10129  ; RK_02 电芯进料机构MES入站读取条码开始字, RK_02 电芯进料机构MES入站读取条码结束字
@BSET(071) &0 E2_1201 E2_1230  ; RK_02 电芯进料机构条码开始字, RK_02 电芯进料机构条码结束字
RSTA(531) W65 &0 &5
RSTA(531) H16 &3 &3
AND=(300) D110 &0  ; 电芯进料扫码数据开始字
AND=L(301) D111 &0
AND=L(301) D113 &0
TIMHX(551) 2800 &5  ; 电芯进料扫码数据初始化延时

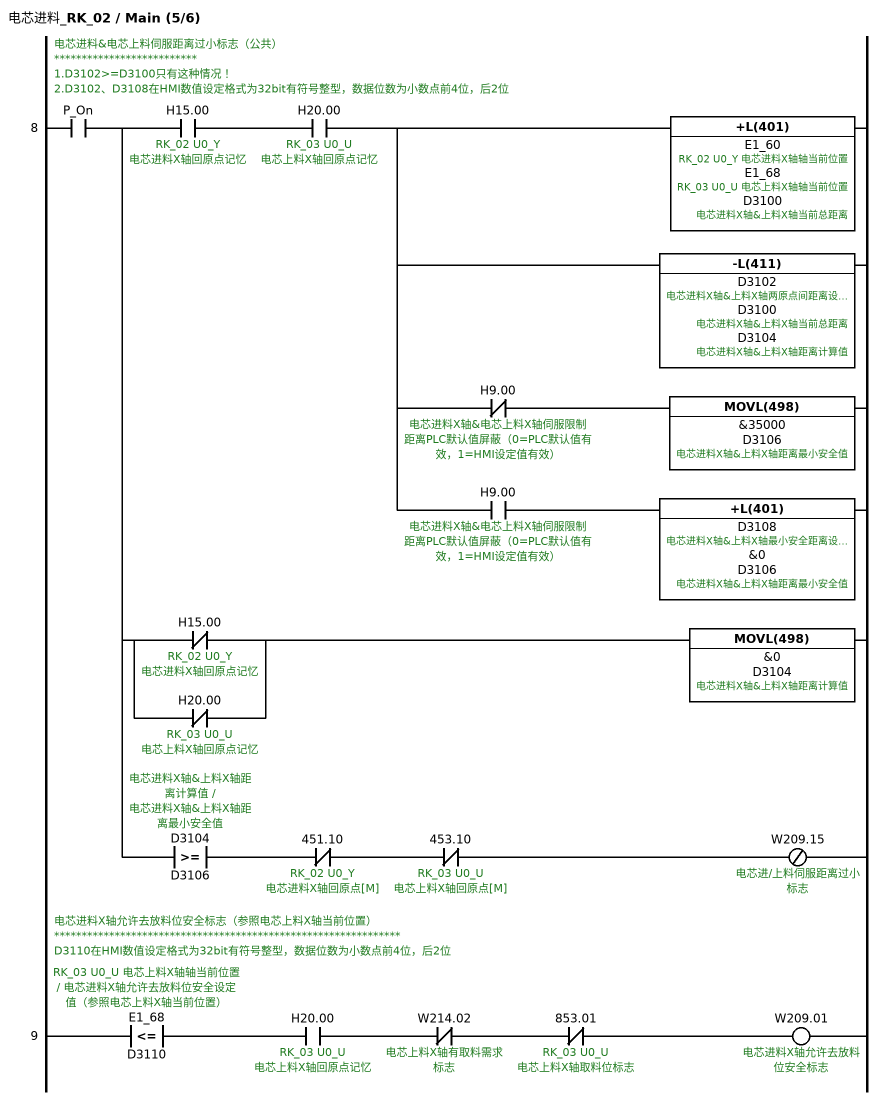
; rung 8: 电芯进料&电芯上料伺服距离过小标志（公共） / ************************** / 1.D3102>=D3100只有这种情况！ / 2.D3102、D3108在HMI数值设定格式为32bit有符号整型，数据位数为小数点前4位，后2位
LD P_On
OUT TR0
AND H15.00  ; RK_02 U0_Y 电芯进料X轴回原点记忆
AND H20.00  ; RK_03 U0_U 电芯上料X轴回原点记忆
OUT TR1
+L(401) E1_60 E1_68 D3100  ; RK_02 U0_Y 电芯进料X轴轴当前位置, RK_03 U0_U 电芯上料X轴轴当前位置, 电芯进料X轴&上料X轴当前总距离
-L(411) D3102 D3100 D3104  ; 电芯进料X轴&上料X轴两原点间距离设定值, 电芯进料X轴&上料X轴当前总距离, 电芯进料X轴&上料X轴距离计算值
ANDNOT H9.00  ; 电芯进料X轴&电芯上料X轴伺服限制距离PLC默认值屏蔽（0=PLC默认值有效，1=HMI设定值有效）
MOVL(498) &35000 D3106  ; 电芯进料X轴&上料X轴距离最小安全值
LD TR1
AND H9.00  ; 电芯进料X轴&电芯上料X轴伺服限制距离PLC默认值屏蔽（0=PLC默认值有效，1=HMI设定值有效）
+L(401) D3108 &0 D3106  ; 电芯进料X轴&上料X轴最小安全距离设定值, 电芯进料X轴&上料X轴距离最小安全值
LD TR0
LDNOT H15.00  ; RK_02 U0_Y 电芯进料X轴回原点记忆
ORNOT H20.00  ; RK_03 U0_U 电芯上料X轴回原点记忆
ANDLD
MOVL(498) &0 D3104  ; 电芯进料X轴&上料X轴距离计算值
LD TR0
AND>=SL(328) D3104 D3106  ; 电芯进料X轴&上料X轴距离计算值, 电芯进料X轴&上料X轴距离最小安全值
ANDNOT 451.10  ; RK_02 U0_Y 电芯进料X轴回原点[M]
ANDNOT 453.10  ; RK_03 U0_U 电芯上料X轴回原点[M]
OUTNOT W209.15  ; 电芯进/上料伺服距离过小标志
; rung 9: 电芯进料X轴允许去放料位安全标志（参照电芯上料X轴当前位置） / *************************************************************** / D3110在HMI数值设定格式为32bit有符号整型，数据位数为小数点前4位，后2位
LD<=SL(318) E1_68 D3110  ; RK_03 U0_U 电芯上料X轴轴当前位置, 电芯进料X轴允许去放料位安全设定值（参照电芯上料X轴当前位置）
AND H20.00  ; RK_03 U0_U 电芯上料X轴回原点记忆
ANDNOT W214.02  ; 电芯上料X轴有取料需求标志
ANDNOT 853.01  ; RK_03 U0_U 电芯上料X轴取料位标志
OUT W209.01  ; 电芯进料X轴允许去放料位安全标志

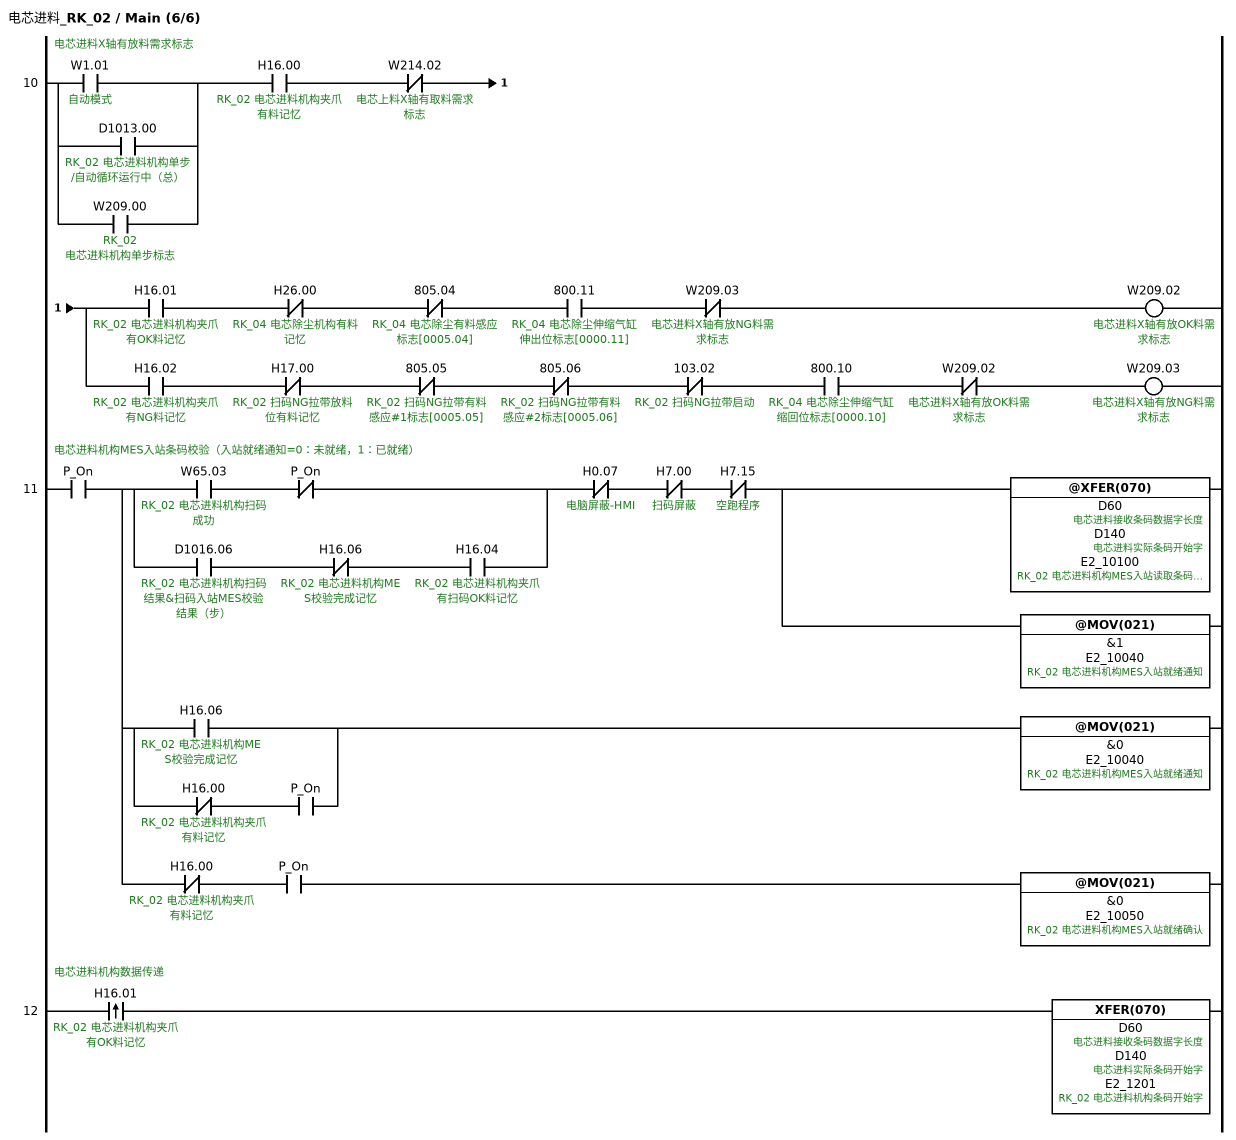
; rung 10: 电芯进料X轴有放料需求标志
LD W1.01  ; 自动模式
OR D1013.00  ; RK_02 电芯进料机构单步/自动循环运行中（总）
OR W209.00  ; RK_02  电芯进料机构单步标志
AND H16.00  ; RK_02 电芯进料机构夹爪有料记忆
ANDNOT W214.02  ; 电芯上料X轴有取料需求标志
OUT TR0
AND H16.01  ; RK_02 电芯进料机构夹爪有OK料记忆
ANDNOT H26.00  ; RK_04 电芯除尘机构有料记忆
ANDNOT 805.04  ; RK_04 电芯除尘有料感应标志[0005.04]
AND 800.11  ; RK_04 电芯除尘伸缩气缸伸出位标志[0000.11]
ANDNOT W209.03  ; 电芯进料X轴有放NG料需求标志
OUT W209.02  ; 电芯进料X轴有放OK料需求标志
LD TR0
AND H16.02  ; RK_02 电芯进料机构夹爪有NG料记忆
ANDNOT H17.00  ; RK_02 扫码NG拉带放料位有料记忆
ANDNOT 805.05  ; RK_02 扫码NG拉带有料感应#1标志[0005.05]
ANDNOT 805.06  ; RK_02 扫码NG拉带有料感应#2标志[0005.06]
ANDNOT 103.02  ; RK_02 扫码NG拉带启动
AND 800.10  ; RK_04 电芯除尘伸缩气缸缩回位标志[0000.10]
ANDNOT W209.02  ; 电芯进料X轴有放OK料需求标志
OUT W209.03  ; 电芯进料X轴有放NG料需求标志
; rung 11: 电芯进料机构MES入站条码校验（入站就绪通知=0：未就绪，1：已就绪）
LD P_On
OUT TR0
LD W65.03  ; RK_02 电芯进料机构扫码成功
ANDNOT P_On
LD D1016.06  ; RK_02 电芯进料机构扫码结果&扫码入站MES校验结果（步）
ANDNOT H16.06  ; RK_02 电芯进料机构MES校验完成记忆
AND H16.04  ; RK_02 电芯进料机构夹爪有扫码OK料记忆
ORLD
ANDLD
ANDNOT H0.07  ; 电脑屏蔽-HMI
ANDNOT H7.00  ; 扫码屏蔽
ANDNOT H7.15  ; 空跑程序
@XFER(070) D60 D140 E2_10100  ; 电芯进料接收条码数据字长度, 电芯进料实际条码开始字, RK_02 电芯进料机构MES入站读取条码开始字
@MOV(021) &1 E2_10040  ; RK_02 电芯进料机构MES入站就绪通知
LD TR0
LD H16.06  ; RK_02 电芯进料机构MES校验完成记忆
LDNOT H16.00  ; RK_02 电芯进料机构夹爪有料记忆
AND P_On
ORLD
ANDLD
@MOV(021) &0 E2_10040  ; RK_02 电芯进料机构MES入站就绪通知
LD TR0
ANDNOT H16.00  ; RK_02 电芯进料机构夹爪有料记忆
AND P_On
@MOV(021) &0 E2_10050  ; RK_02 电芯进料机构MES入站就绪确认
; rung 12: 电芯进料机构数据传递
@LD H16.01  ; RK_02 电芯进料机构夹爪有OK料记忆
XFER(070) D60 D140 E2_1201  ; 电芯进料接收条码数据字长度, 电芯进料实际条码开始字, RK_02 电芯进料机构条码开始字

### Section 手动

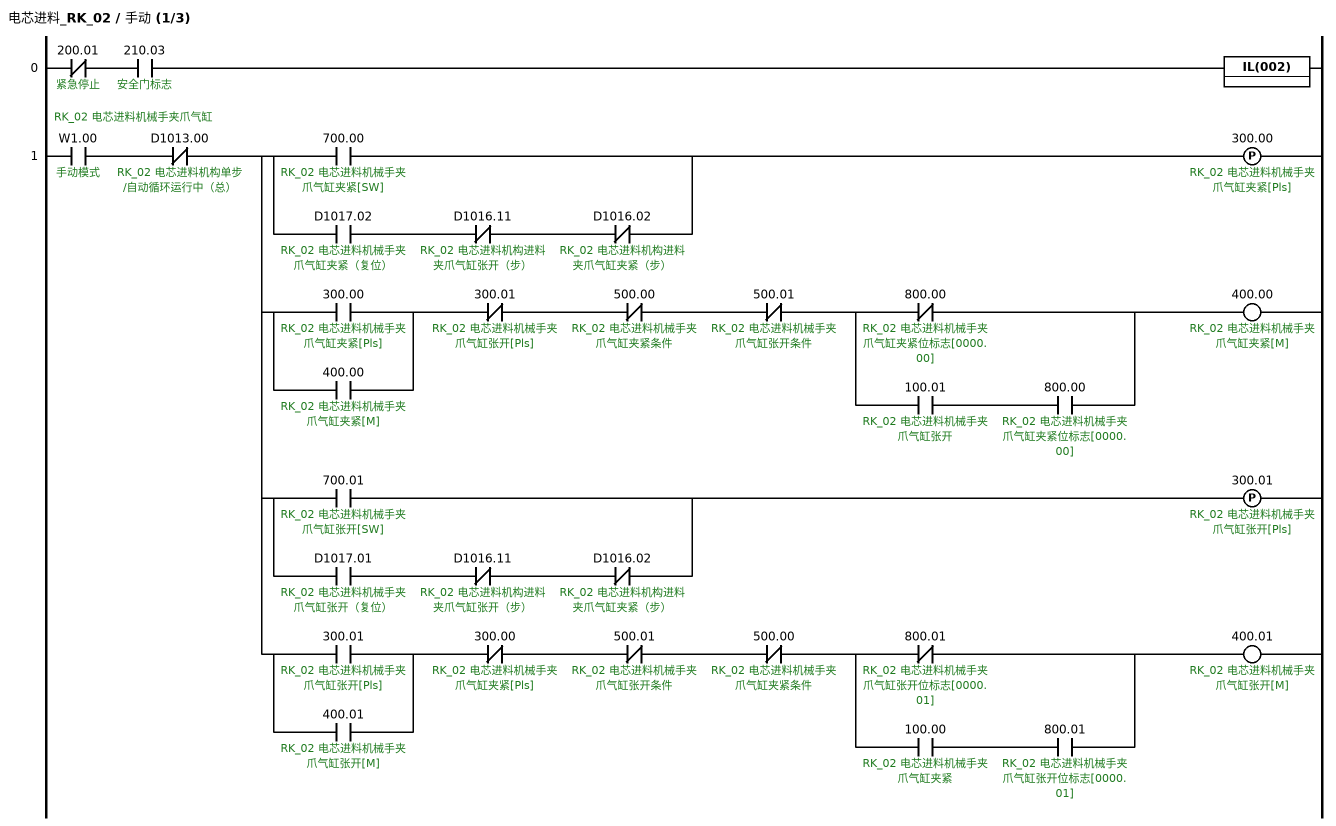
; rung 0
LDNOT 200.01  ; 紧急停止
AND 210.03  ; 安全门标志
IL(002)
; rung 1: RK_02 电芯进料机械手夹爪气缸
LD W1.00  ; 手动模式
ANDNOT D1013.00  ; RK_02 电芯进料机构单步/自动循环运行中（总）
OUT TR0
LD 700.00  ; RK_02 电芯进料机械手夹爪气缸夹紧[SW]
LD D1017.02  ; RK_02 电芯进料机械手夹爪气缸夹紧（复位）
ANDNOT D1016.11  ; RK_02 电芯进料机构进料夹爪气缸张开（步）
ANDNOT D1016.02  ; RK_02 电芯进料机构进料夹爪气缸夹紧（步）
ORLD
ANDLD
DIFU(013) 300.00  ; RK_02 电芯进料机械手夹爪气缸夹紧[Pls]
LD TR0
LD 300.00  ; RK_02 电芯进料机械手夹爪气缸夹紧[Pls]
OR 400.00  ; RK_02 电芯进料机械手夹爪气缸夹紧[M]
ANDLD
ANDNOT 300.01  ; RK_02 电芯进料机械手夹爪气缸张开[Pls]
ANDNOT 500.00  ; RK_02 电芯进料机械手夹爪气缸夹紧条件
ANDNOT 500.01  ; RK_02 电芯进料机械手夹爪气缸张开条件
LDNOT 800.00  ; RK_02 电芯进料机械手夹爪气缸夹紧位标志[0000.00]
LD 100.01  ; RK_02 电芯进料机械手夹爪气缸张开
AND 800.00  ; RK_02 电芯进料机械手夹爪气缸夹紧位标志[0000.00]
ORLD
ANDLD
OUT 400.00  ; RK_02 电芯进料机械手夹爪气缸夹紧[M]
LD TR0
LD 700.01  ; RK_02 电芯进料机械手夹爪气缸张开[SW]
LD D1017.01  ; RK_02 电芯进料机械手夹爪气缸张开（复位）
ANDNOT D1016.11  ; RK_02 电芯进料机构进料夹爪气缸张开（步）
ANDNOT D1016.02  ; RK_02 电芯进料机构进料夹爪气缸夹紧（步）
ORLD
ANDLD
DIFU(013) 300.01  ; RK_02 电芯进料机械手夹爪气缸张开[Pls]
LD TR0
LD 300.01  ; RK_02 电芯进料机械手夹爪气缸张开[Pls]
OR 400.01  ; RK_02 电芯进料机械手夹爪气缸张开[M]
ANDLD
ANDNOT 300.00  ; RK_02 电芯进料机械手夹爪气缸夹紧[Pls]
ANDNOT 500.01  ; RK_02 电芯进料机械手夹爪气缸张开条件
ANDNOT 500.00  ; RK_02 电芯进料机械手夹爪气缸夹紧条件
LDNOT 800.01  ; RK_02 电芯进料机械手夹爪气缸张开位标志[0000.01]
LD 100.00  ; RK_02 电芯进料机械手夹爪气缸夹紧
AND 800.01  ; RK_02 电芯进料机械手夹爪气缸张开位标志[0000.01]
ORLD
ANDLD
OUT 400.01  ; RK_02 电芯进料机械手夹爪气缸张开[M]

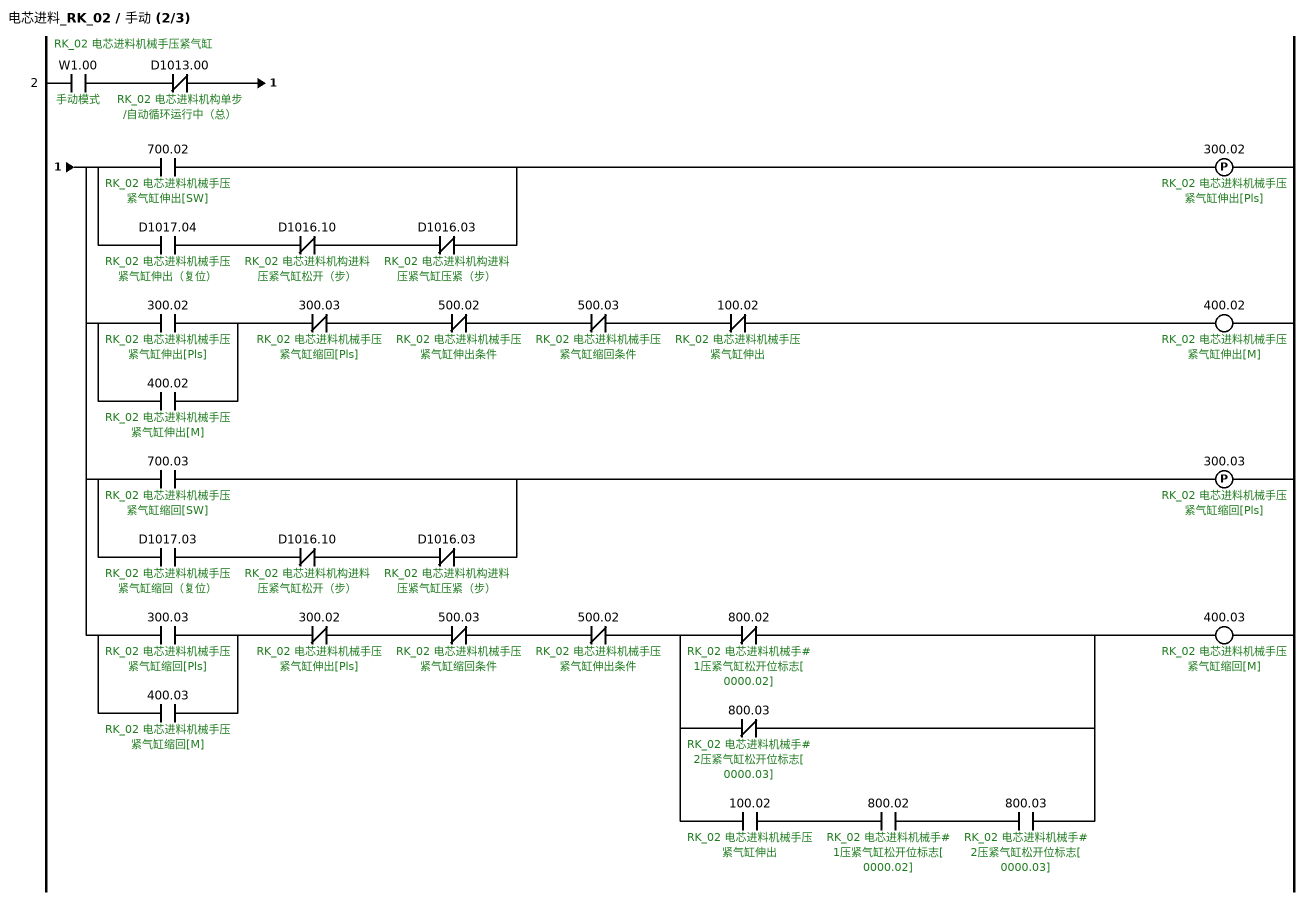
; rung 2: RK_02 电芯进料机械手压紧气缸
LD W1.00  ; 手动模式
ANDNOT D1013.00  ; RK_02 电芯进料机构单步/自动循环运行中（总）
OUT TR0
LD 700.02  ; RK_02 电芯进料机械手压紧气缸伸出[SW]
LD D1017.04  ; RK_02 电芯进料机械手压紧气缸伸出（复位）
ANDNOT D1016.10  ; RK_02 电芯进料机构进料压紧气缸松开（步）
ANDNOT D1016.03  ; RK_02 电芯进料机构进料压紧气缸压紧（步）
ORLD
ANDLD
DIFU(013) 300.02  ; RK_02 电芯进料机械手压紧气缸伸出[Pls]
LD TR0
LD 300.02  ; RK_02 电芯进料机械手压紧气缸伸出[Pls]
OR 400.02  ; RK_02 电芯进料机械手压紧气缸伸出[M]
ANDLD
ANDNOT 300.03  ; RK_02 电芯进料机械手压紧气缸缩回[Pls]
ANDNOT 500.02  ; RK_02 电芯进料机械手压紧气缸伸出条件
ANDNOT 500.03  ; RK_02 电芯进料机械手压紧气缸缩回条件
ANDNOT 100.02  ; RK_02 电芯进料机械手压紧气缸伸出
OUT 400.02  ; RK_02 电芯进料机械手压紧气缸伸出[M]
LD TR0
LD 700.03  ; RK_02 电芯进料机械手压紧气缸缩回[SW]
LD D1017.03  ; RK_02 电芯进料机械手压紧气缸缩回（复位）
ANDNOT D1016.10  ; RK_02 电芯进料机构进料压紧气缸松开（步）
ANDNOT D1016.03  ; RK_02 电芯进料机构进料压紧气缸压紧（步）
ORLD
ANDLD
DIFU(013) 300.03  ; RK_02 电芯进料机械手压紧气缸缩回[Pls]
LD TR0
LD 300.03  ; RK_02 电芯进料机械手压紧气缸缩回[Pls]
OR 400.03  ; RK_02 电芯进料机械手压紧气缸缩回[M]
ANDLD
ANDNOT 300.02  ; RK_02 电芯进料机械手压紧气缸伸出[Pls]
ANDNOT 500.03  ; RK_02 电芯进料机械手压紧气缸缩回条件
ANDNOT 500.02  ; RK_02 电芯进料机械手压紧气缸伸出条件
LDNOT 800.02  ; RK_02 电芯进料机械手#1压紧气缸松开位标志[0000.02]
ORNOT 800.03  ; RK_02 电芯进料机械手#2压紧气缸松开位标志[0000.03]
LD 100.02  ; RK_02 电芯进料机械手压紧气缸伸出
AND 800.02  ; RK_02 电芯进料机械手#1压紧气缸松开位标志[0000.02]
AND 800.03  ; RK_02 电芯进料机械手#2压紧气缸松开位标志[0000.03]
ORLD
ANDLD
OUT 400.03  ; RK_02 电芯进料机械手压紧气缸缩回[M]

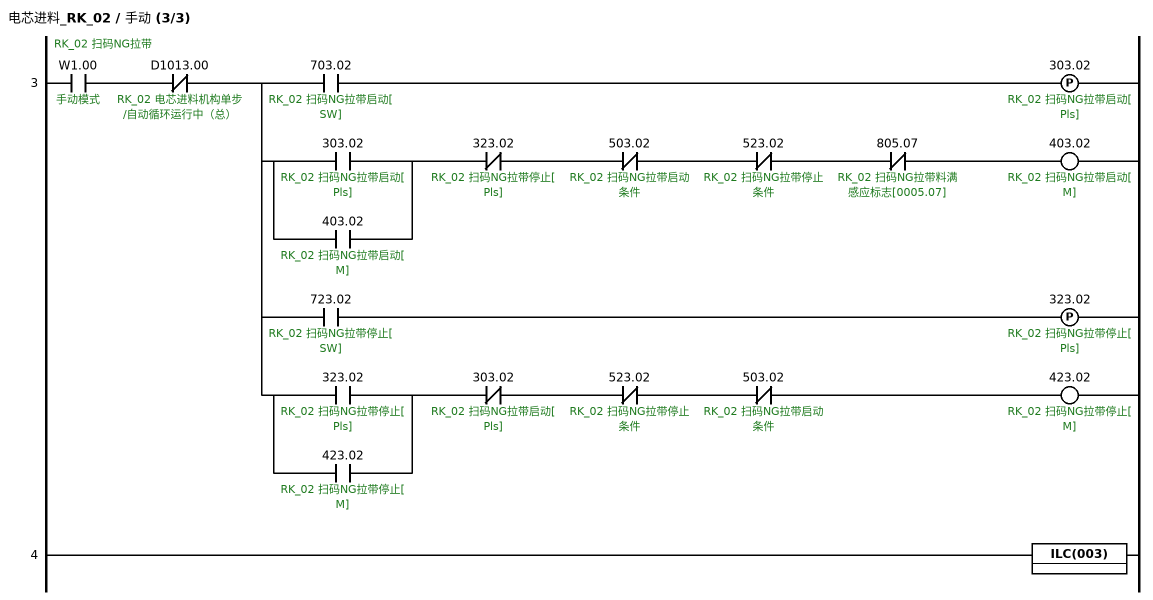
; rung 3: RK_02 扫码NG拉带
LD W1.00  ; 手动模式
ANDNOT D1013.00  ; RK_02 电芯进料机构单步/自动循环运行中（总）
OUT TR0
AND 703.02  ; RK_02 扫码NG拉带启动[SW]
DIFU(013) 303.02  ; RK_02 扫码NG拉带启动[Pls]
LD TR0
LD 303.02  ; RK_02 扫码NG拉带启动[Pls]
OR 403.02  ; RK_02 扫码NG拉带启动[M]
ANDLD
ANDNOT 323.02  ; RK_02 扫码NG拉带停止[Pls]
ANDNOT 503.02  ; RK_02 扫码NG拉带启动条件
ANDNOT 523.02  ; RK_02 扫码NG拉带停止条件
ANDNOT 805.07  ; RK_02 扫码NG拉带料满感应标志[0005.07]
OUT 403.02  ; RK_02 扫码NG拉带启动[M]
LD TR0
AND 723.02  ; RK_02 扫码NG拉带停止[SW]
DIFU(013) 323.02  ; RK_02 扫码NG拉带停止[Pls]
LD TR0
LD 323.02  ; RK_02 扫码NG拉带停止[Pls]
OR 423.02  ; RK_02 扫码NG拉带停止[M]
ANDLD
ANDNOT 303.02  ; RK_02 扫码NG拉带启动[Pls]
ANDNOT 523.02  ; RK_02 扫码NG拉带停止条件
ANDNOT 503.02  ; RK_02 扫码NG拉带启动条件
OUT 423.02  ; RK_02 扫码NG拉带停止[M]
; rung 4
ILC(003)

### Section 自动

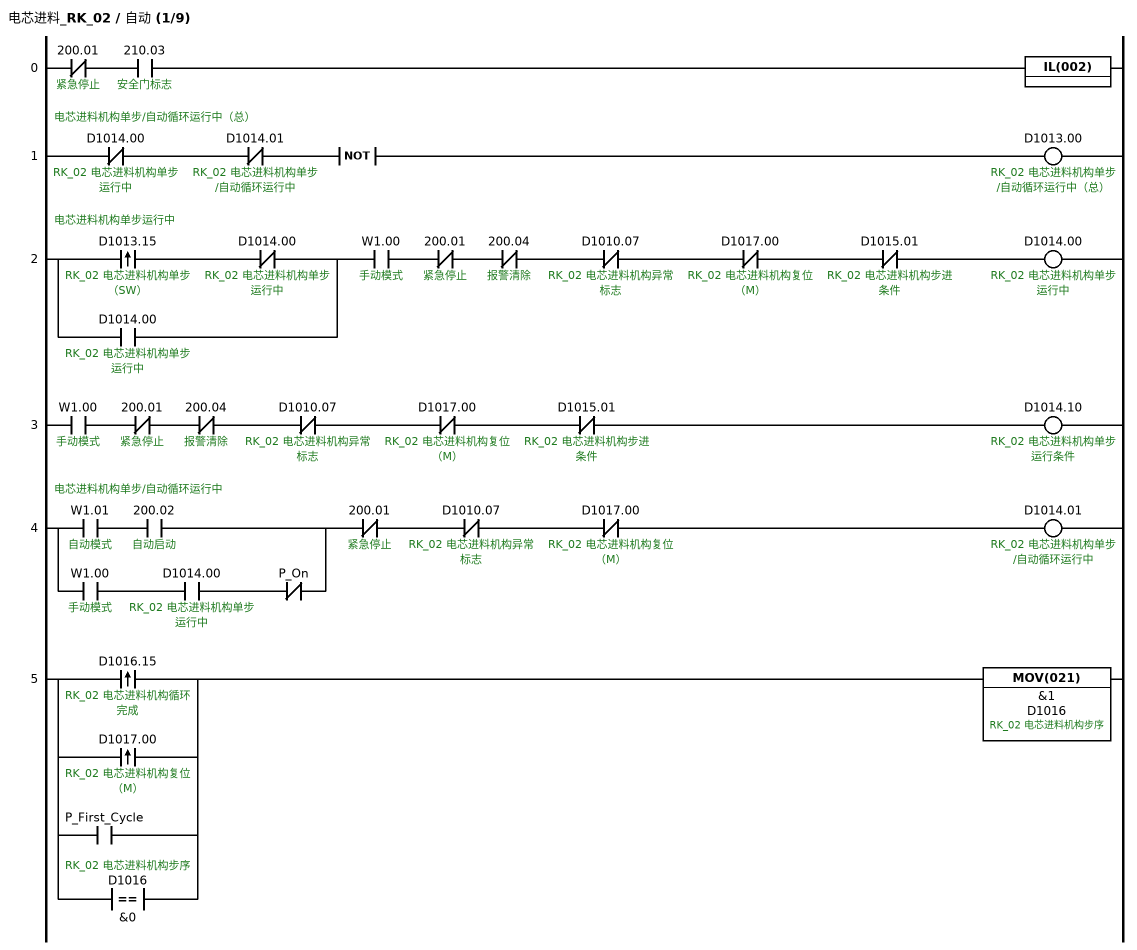
; rung 0
LDNOT 200.01  ; 紧急停止
AND 210.03  ; 安全门标志
IL(002)
; rung 1: 电芯进料机构单步/自动循环运行中（总）
LDNOT D1014.00  ; RK_02 电芯进料机构单步运行中
ANDNOT D1014.01  ; RK_02 电芯进料机构单步/自动循环运行中
NOT(520)
OUT D1013.00  ; RK_02 电芯进料机构单步/自动循环运行中（总）
; rung 2: 电芯进料机构单步运行中
@LD D1013.15  ; RK_02 电芯进料机构单步（SW）
ANDNOT D1014.00  ; RK_02 电芯进料机构单步运行中
OR D1014.00  ; RK_02 电芯进料机构单步运行中
AND W1.00  ; 手动模式
ANDNOT 200.01  ; 紧急停止
ANDNOT 200.04  ; 报警清除
ANDNOT D1010.07  ; RK_02 电芯进料机构异常标志
ANDNOT D1017.00  ; RK_02 电芯进料机构复位（M）
ANDNOT D1015.01  ; RK_02 电芯进料机构步进条件
OUT D1014.00  ; RK_02 电芯进料机构单步运行中
; rung 3
LD W1.00  ; 手动模式
ANDNOT 200.01  ; 紧急停止
ANDNOT 200.04  ; 报警清除
ANDNOT D1010.07  ; RK_02 电芯进料机构异常标志
ANDNOT D1017.00  ; RK_02 电芯进料机构复位（M）
ANDNOT D1015.01  ; RK_02 电芯进料机构步进条件
OUT D1014.10  ; RK_02 电芯进料机构单步运行条件
; rung 4: 电芯进料机构单步/自动循环运行中
LD W1.01  ; 自动模式
AND 200.02  ; 自动启动
LD W1.00  ; 手动模式
AND D1014.00  ; RK_02 电芯进料机构单步运行中
ANDNOT P_On
ORLD
ANDNOT 200.01  ; 紧急停止
ANDNOT D1010.07  ; RK_02 电芯进料机构异常标志
ANDNOT D1017.00  ; RK_02 电芯进料机构复位（M）
OUT D1014.01  ; RK_02 电芯进料机构单步/自动循环运行中
; rung 5
@LD D1016.15  ; RK_02 电芯进料机构循环完成
@OR D1017.00  ; RK_02 电芯进料机构复位（M）
OR P_First_Cycle
OR=(300) D1016 &0  ; RK_02 电芯进料机构步序
MOV(021) &1 D1016  ; RK_02 电芯进料机构步序

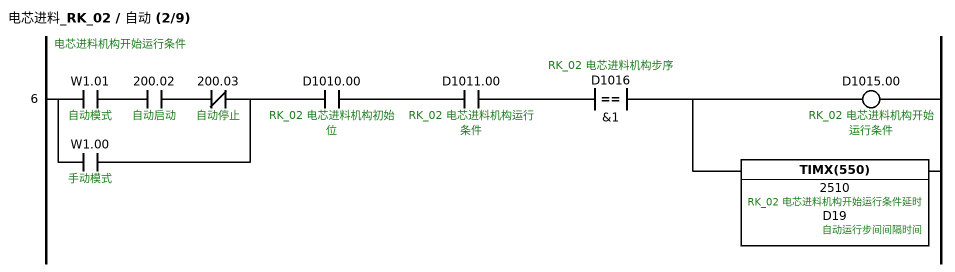
; rung 6: 电芯进料机构开始运行条件
LD W1.01  ; 自动模式
AND 200.02  ; 自动启动
ANDNOT 200.03  ; 自动停止
OR W1.00  ; 手动模式
AND D1010.00  ; RK_02 电芯进料机构初始位
AND D1011.00  ; RK_02 电芯进料机构运行条件
AND=(300) D1016 &1  ; RK_02 电芯进料机构步序
OUT D1015.00  ; RK_02 电芯进料机构开始运行条件
TIMX(550) 2510 D19  ; 自动运行步间间隔时间, RK_02 电芯进料机构开始运行条件延时

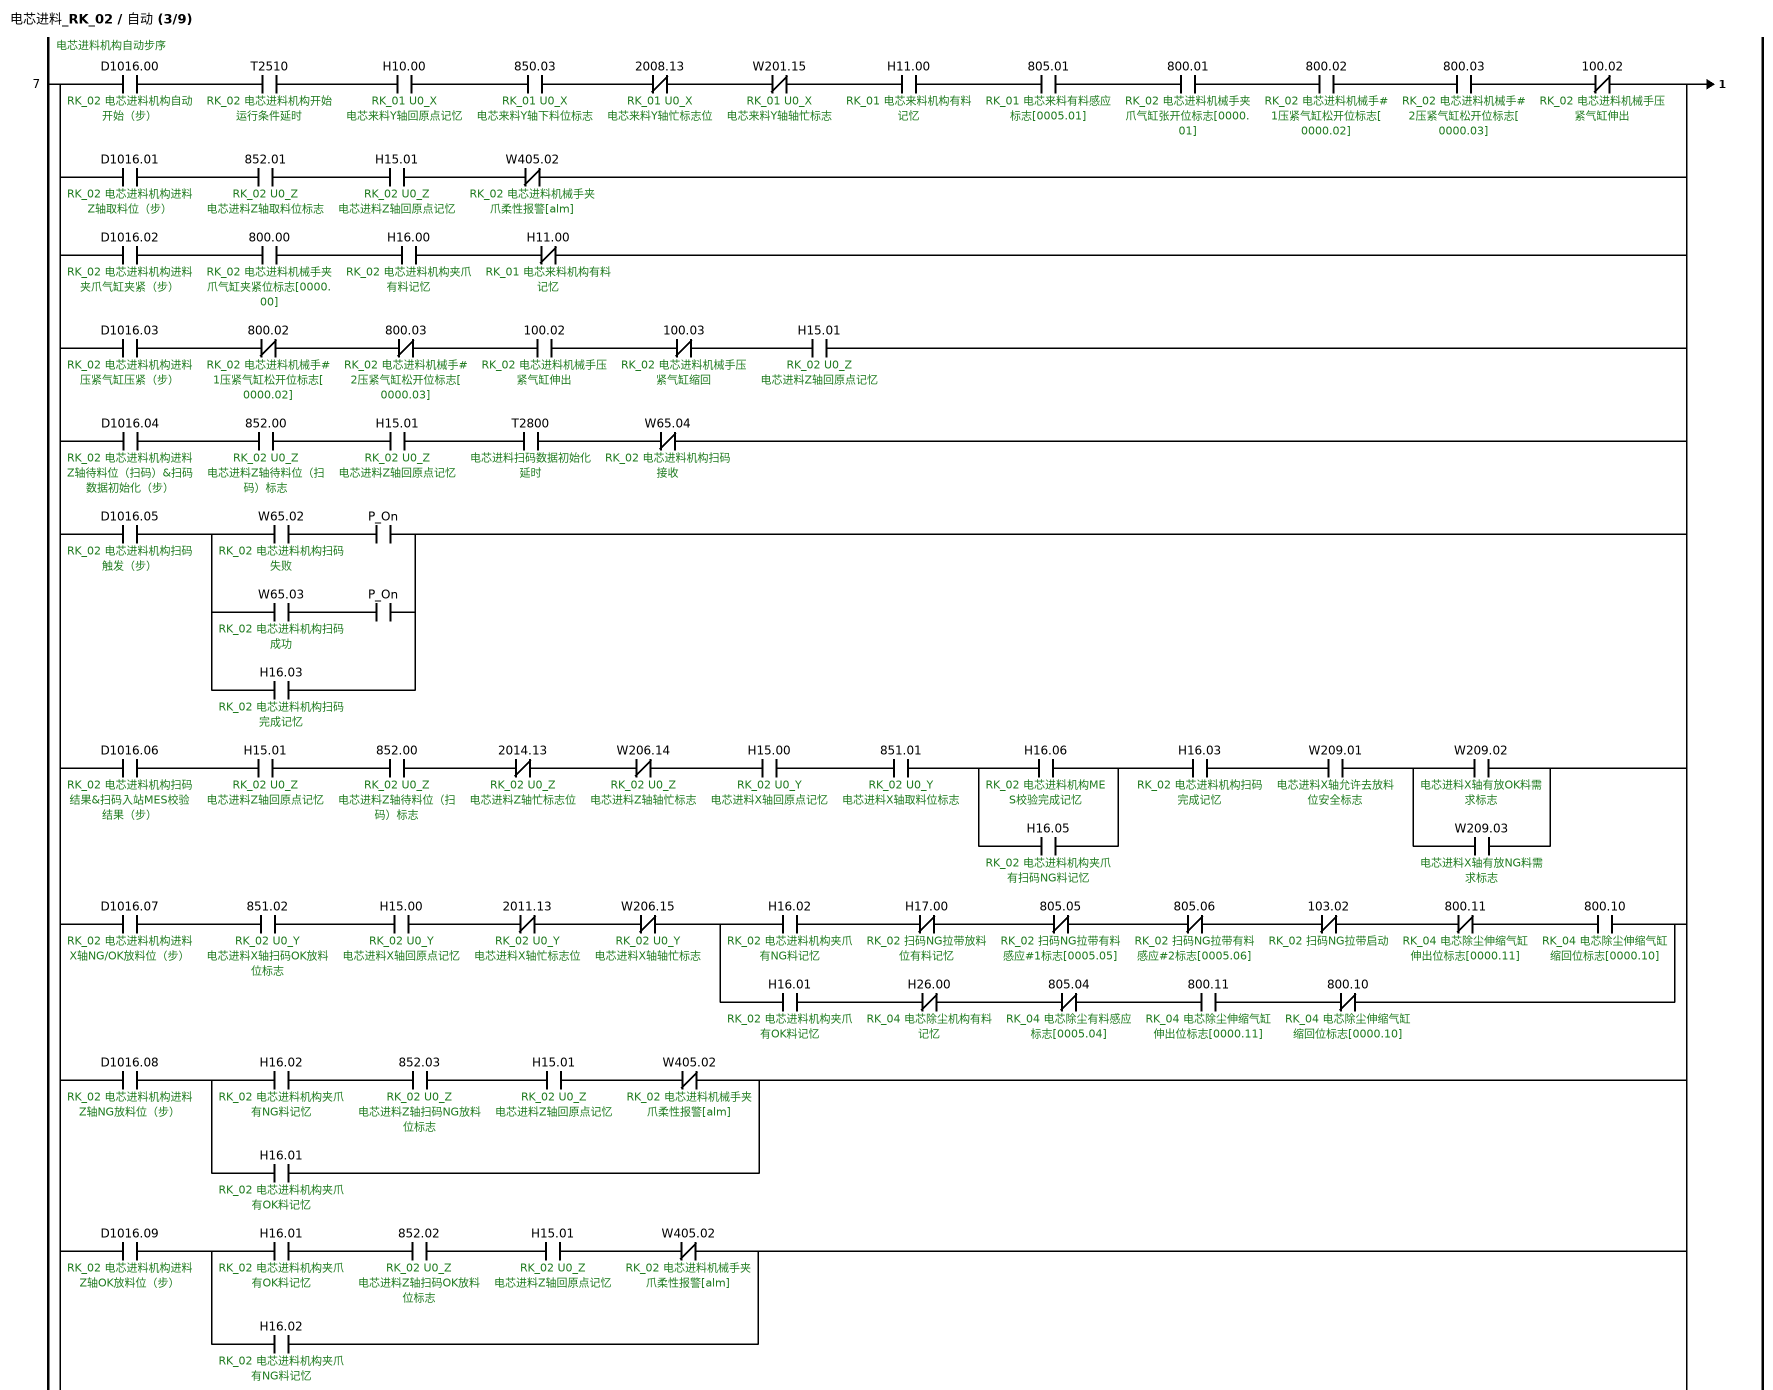

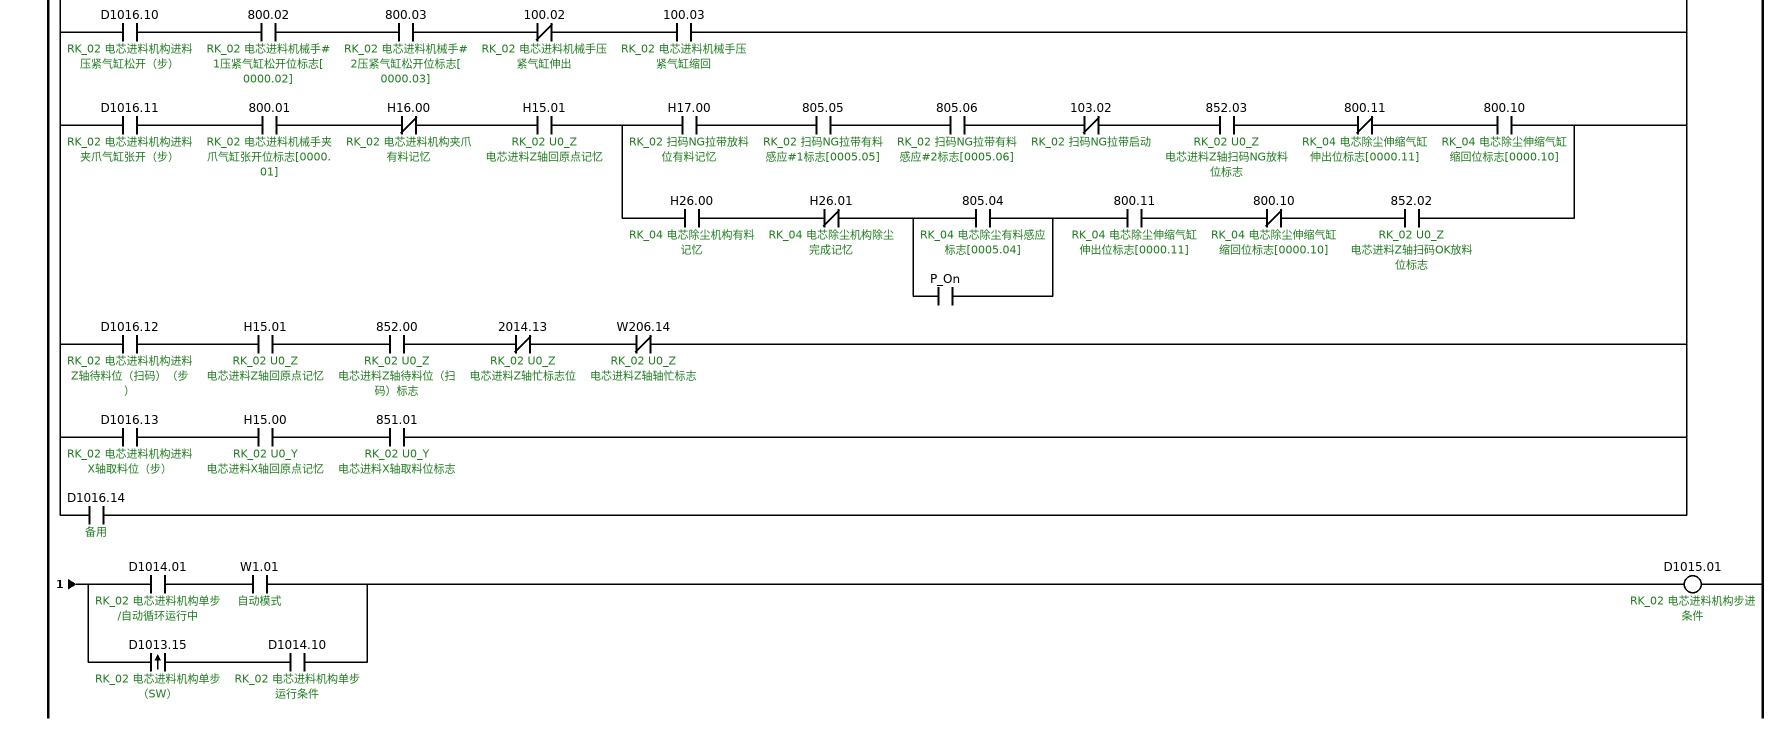
; rung 7: 电芯进料机构自动步序
LD D1016.00  ; RK_02 电芯进料机构自动开始（步）
AND T2510  ; RK_02 电芯进料机构开始运行条件延时
AND H10.00  ; RK_01 U0_X 电芯来料Y轴回原点记忆
AND 850.03  ; RK_01 U0_X 电芯来料Y轴下料位标志
ANDNOT 2008.13  ; RK_01 U0_X 电芯来料Y轴忙标志位
ANDNOT W201.15  ; RK_01 U0_X 电芯来料Y轴轴忙标志
AND H11.00  ; RK_01 电芯来料机构有料记忆
AND 805.01  ; RK_01 电芯来料有料感应标志[0005.01]
AND 800.01  ; RK_02 电芯进料机械手夹爪气缸张开位标志[0000.01]
AND 800.02  ; RK_02 电芯进料机械手#1压紧气缸松开位标志[0000.02]
AND 800.03  ; RK_02 电芯进料机械手#2压紧气缸松开位标志[0000.03]
ANDNOT 100.02  ; RK_02 电芯进料机械手压紧气缸伸出
LD D1016.01  ; RK_02 电芯进料机构进料Z轴取料位（步）
AND 852.01  ; RK_02 U0_Z 电芯进料Z轴取料位标志
AND H15.01  ; RK_02 U0_Z 电芯进料Z轴回原点记忆
ANDNOT W405.02  ; RK_02 电芯进料机械手夹爪柔性报警[alm]
ORLD
LD D1016.02  ; RK_02 电芯进料机构进料夹爪气缸夹紧（步）
AND 800.00  ; RK_02 电芯进料机械手夹爪气缸夹紧位标志[0000.00]
AND H16.00  ; RK_02 电芯进料机构夹爪有料记忆
ANDNOT H11.00  ; RK_01 电芯来料机构有料记忆
ORLD
LD D1016.03  ; RK_02 电芯进料机构进料压紧气缸压紧（步）
ANDNOT 800.02  ; RK_02 电芯进料机械手#1压紧气缸松开位标志[0000.02]
ANDNOT 800.03  ; RK_02 电芯进料机械手#2压紧气缸松开位标志[0000.03]
AND 100.02  ; RK_02 电芯进料机械手压紧气缸伸出
ANDNOT 100.03  ; RK_02 电芯进料机械手压紧气缸缩回
AND H15.01  ; RK_02 U0_Z 电芯进料Z轴回原点记忆
ORLD
LD D1016.04  ; RK_02 电芯进料机构进料Z轴待料位（扫码）&扫码数据初始化（步）
AND 852.00  ; RK_02 U0_Z 电芯进料Z轴待料位（扫码）标志
AND H15.01  ; RK_02 U0_Z 电芯进料Z轴回原点记忆
AND T2800  ; 电芯进料扫码数据初始化延时
ANDNOT W65.04  ; RK_02 电芯进料机构扫码接收
ORLD
LD D1016.05  ; RK_02 电芯进料机构扫码触发（步）
LD W65.02  ; RK_02 电芯进料机构扫码失败
AND P_On
LD W65.03  ; RK_02 电芯进料机构扫码成功
AND P_On
ORLD
OR H16.03  ; RK_02 电芯进料机构扫码完成记忆
ANDLD
ORLD
LD D1016.06  ; RK_02 电芯进料机构扫码结果&扫码入站MES校验结果（步）
AND H15.01  ; RK_02 U0_Z 电芯进料Z轴回原点记忆
AND 852.00  ; RK_02 U0_Z 电芯进料Z轴待料位（扫码）标志
ANDNOT 2014.13  ; RK_02 U0_Z 电芯进料Z轴忙标志位
ANDNOT W206.14  ; RK_02 U0_Z 电芯进料Z轴轴忙标志
AND H15.00  ; RK_02 U0_Y 电芯进料X轴回原点记忆
AND 851.01  ; RK_02 U0_Y 电芯进料X轴取料位标志
LD H16.06  ; RK_02 电芯进料机构MES校验完成记忆
OR H16.05  ; RK_02 电芯进料机构夹爪有扫码NG料记忆
ANDLD
AND H16.03  ; RK_02 电芯进料机构扫码完成记忆
AND W209.01  ; 电芯进料X轴允许去放料位安全标志
LD W209.02  ; 电芯进料X轴有放OK料需求标志
OR W209.03  ; 电芯进料X轴有放NG料需求标志
ANDLD
ORLD
LD D1016.07  ; RK_02 电芯进料机构进料X轴NG/OK放料位（步）
AND 851.02  ; RK_02 U0_Y 电芯进料X轴扫码OK放料位标志
AND H15.00  ; RK_02 U0_Y 电芯进料X轴回原点记忆
ANDNOT 2011.13  ; RK_02 U0_Y 电芯进料X轴忙标志位
ANDNOT W206.15  ; RK_02 U0_Y 电芯进料X轴轴忙标志
LD H16.02  ; RK_02 电芯进料机构夹爪有NG料记忆
ANDNOT H17.00  ; RK_02 扫码NG拉带放料位有料记忆
ANDNOT 805.05  ; RK_02 扫码NG拉带有料感应#1标志[0005.05]
ANDNOT 805.06  ; RK_02 扫码NG拉带有料感应#2标志[0005.06]
ANDNOT 103.02  ; RK_02 扫码NG拉带启动
ANDNOT 800.11  ; RK_04 电芯除尘伸缩气缸伸出位标志[0000.11]
AND 800.10  ; RK_04 电芯除尘伸缩气缸缩回位标志[0000.10]
LD H16.01  ; RK_02 电芯进料机构夹爪有OK料记忆
ANDNOT H26.00  ; RK_04 电芯除尘机构有料记忆
ANDNOT 805.04  ; RK_04 电芯除尘有料感应标志[0005.04]
AND 800.11  ; RK_04 电芯除尘伸缩气缸伸出位标志[0000.11]
ANDNOT 800.10  ; RK_04 电芯除尘伸缩气缸缩回位标志[0000.10]
ORLD
ANDLD
ORLD
LD D1016.08  ; RK_02 电芯进料机构进料Z轴NG放料位（步）
LD H16.02  ; RK_02 电芯进料机构夹爪有NG料记忆
AND 852.03  ; RK_02 U0_Z 电芯进料Z轴扫码NG放料位标志
AND H15.01  ; RK_02 U0_Z 电芯进料Z轴回原点记忆
ANDNOT W405.02  ; RK_02 电芯进料机械手夹爪柔性报警[alm]
OR H16.01  ; RK_02 电芯进料机构夹爪有OK料记忆
ANDLD
ORLD
LD D1016.09  ; RK_02 电芯进料机构进料Z轴OK放料位（步）
LD H16.01  ; RK_02 电芯进料机构夹爪有OK料记忆
AND 852.02  ; RK_02 U0_Z 电芯进料Z轴扫码OK放料位标志
AND H15.01  ; RK_02 U0_Z 电芯进料Z轴回原点记忆
ANDNOT W405.02  ; RK_02 电芯进料机械手夹爪柔性报警[alm]
OR H16.02  ; RK_02 电芯进料机构夹爪有NG料记忆
ANDLD
ORLD
LD D1016.10  ; RK_02 电芯进料机构进料压紧气缸松开（步）
AND 800.02  ; RK_02 电芯进料机械手#1压紧气缸松开位标志[0000.02]
AND 800.03  ; RK_02 电芯进料机械手#2压紧气缸松开位标志[0000.03]
ANDNOT 100.02  ; RK_02 电芯进料机械手压紧气缸伸出
AND 100.03  ; RK_02 电芯进料机械手压紧气缸缩回
ORLD
LD D1016.11  ; RK_02 电芯进料机构进料夹爪气缸张开（步）
AND 800.01  ; RK_02 电芯进料机械手夹爪气缸张开位标志[0000.01]
ANDNOT H16.00  ; RK_02 电芯进料机构夹爪有料记忆
AND H15.01  ; RK_02 U0_Z 电芯进料Z轴回原点记忆
LD H17.00  ; RK_02 扫码NG拉带放料位有料记忆
AND 805.05  ; RK_02 扫码NG拉带有料感应#1标志[0005.05]
AND 805.06  ; RK_02 扫码NG拉带有料感应#2标志[0005.06]
ANDNOT 103.02  ; RK_02 扫码NG拉带启动
AND 852.03  ; RK_02 U0_Z 电芯进料Z轴扫码NG放料位标志
ANDNOT 800.11  ; RK_04 电芯除尘伸缩气缸伸出位标志[0000.11]
AND 800.10  ; RK_04 电芯除尘伸缩气缸缩回位标志[0000.10]
LD H26.00  ; RK_04 电芯除尘机构有料记忆
ANDNOT H26.01  ; RK_04 电芯除尘机构除尘完成记忆
LD 805.04  ; RK_04 电芯除尘有料感应标志[0005.04]
OR P_On
ANDLD
AND 800.11  ; RK_04 电芯除尘伸缩气缸伸出位标志[0000.11]
ANDNOT 800.10  ; RK_04 电芯除尘伸缩气缸缩回位标志[0000.10]
AND 852.02  ; RK_02 U0_Z 电芯进料Z轴扫码OK放料位标志
ORLD
ANDLD
ORLD
LD D1016.12  ; RK_02 电芯进料机构进料Z轴待料位（扫码）（步）
AND H15.01  ; RK_02 U0_Z 电芯进料Z轴回原点记忆
AND 852.00  ; RK_02 U0_Z 电芯进料Z轴待料位（扫码）标志
ANDNOT 2014.13  ; RK_02 U0_Z 电芯进料Z轴忙标志位
ANDNOT W206.14  ; RK_02 U0_Z 电芯进料Z轴轴忙标志
ORLD
LD D1016.13  ; RK_02 电芯进料机构进料X轴取料位（步）
AND H15.00  ; RK_02 U0_Y 电芯进料X轴回原点记忆
AND 851.01  ; RK_02 U0_Y 电芯进料X轴取料位标志
ORLD
OR D1016.14  ; 备用
LD D1014.01  ; RK_02 电芯进料机构单步/自动循环运行中
AND W1.01  ; 自动模式
@LD D1013.15  ; RK_02 电芯进料机构单步（SW）
AND D1014.10  ; RK_02 电芯进料机构单步运行条件
ORLD
ANDLD
OUT D1015.01  ; RK_02 电芯进料机构步进条件

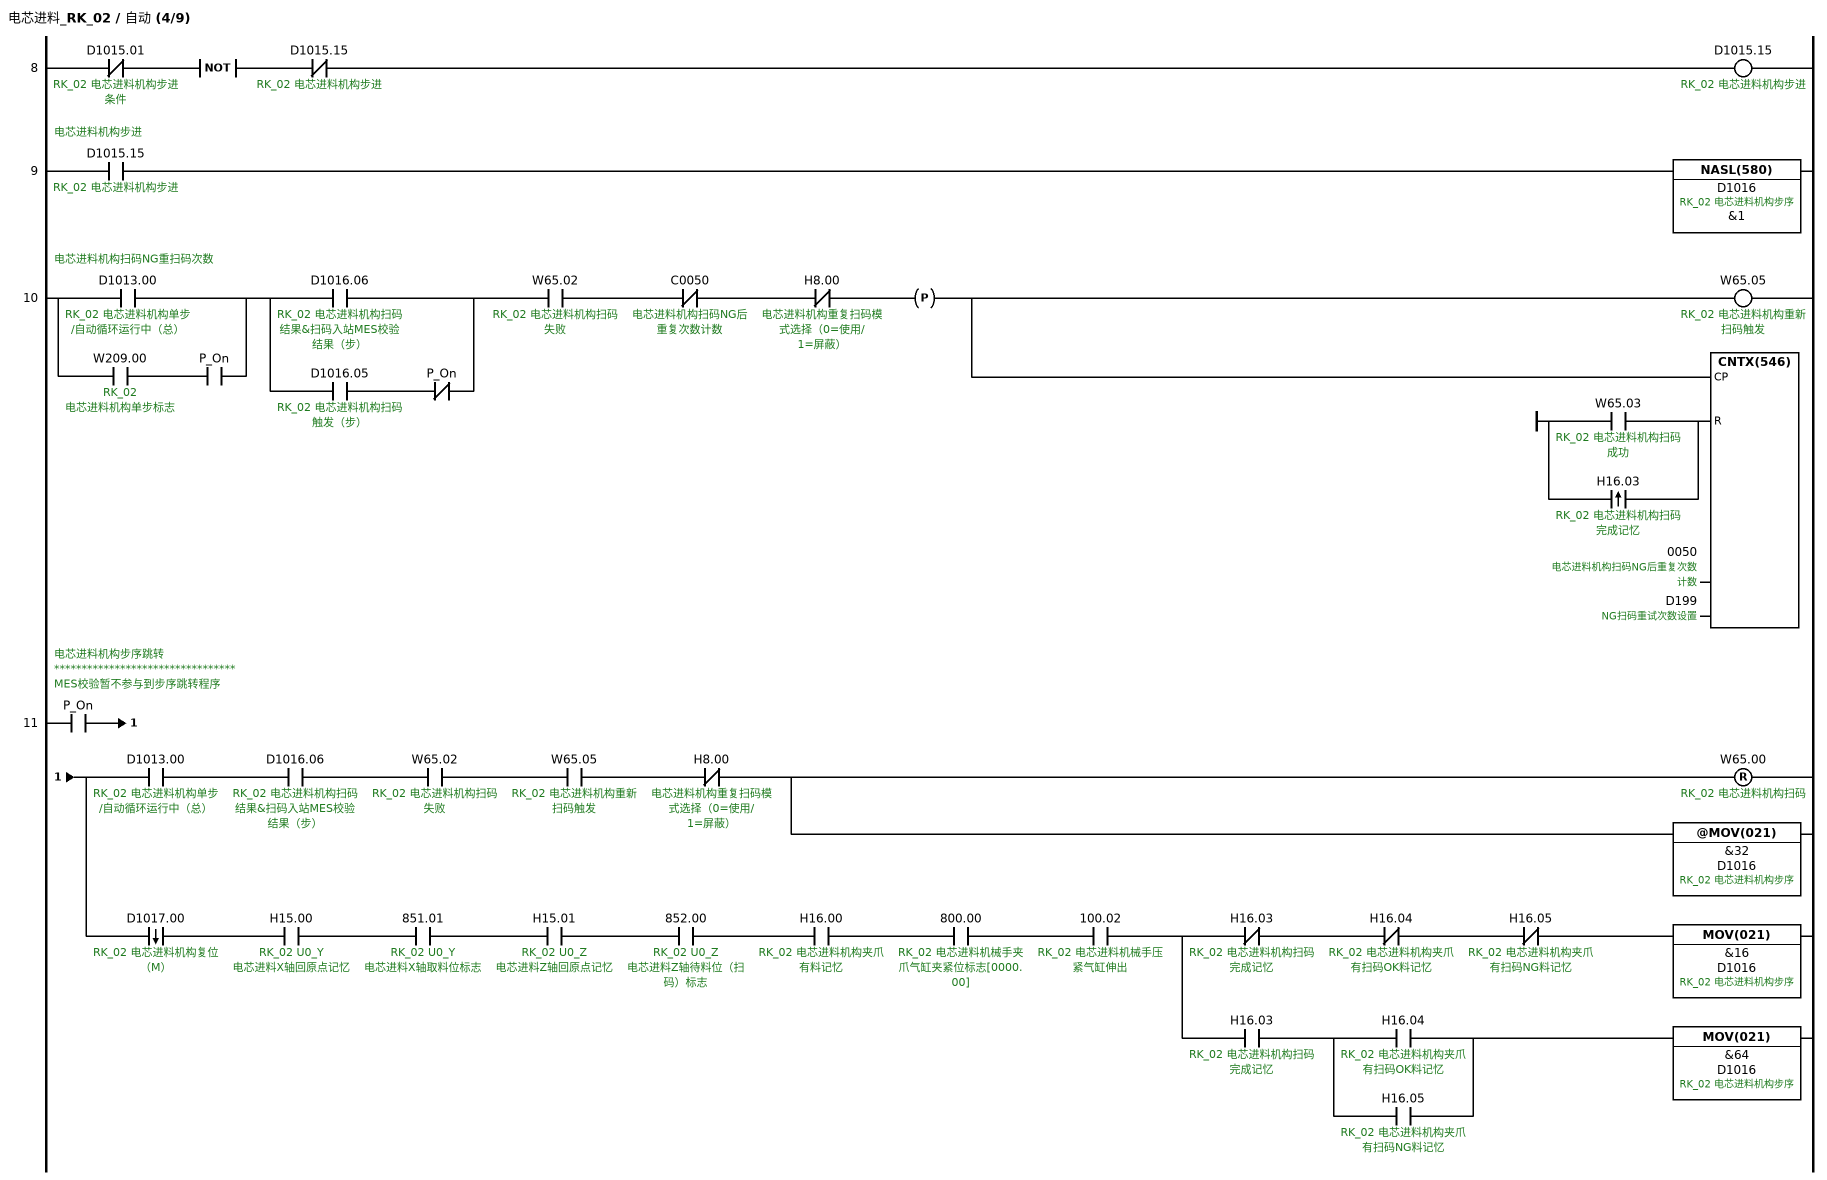
; rung 8
LDNOT D1015.01  ; RK_02 电芯进料机构步进条件
NOT(520)
ANDNOT D1015.15  ; RK_02 电芯进料机构步进
OUT D1015.15  ; RK_02 电芯进料机构步进
; rung 9: 电芯进料机构步进
LD D1015.15  ; RK_02 电芯进料机构步进
NASL(580) D1016 &1  ; RK_02 电芯进料机构步序
; rung 10: 电芯进料机构扫码NG重扫码次数
LD D1013.00  ; RK_02 电芯进料机构单步/自动循环运行中（总）
LD W209.00  ; RK_02  电芯进料机构单步标志
AND P_On
ORLD
LD D1016.06  ; RK_02 电芯进料机构扫码结果&扫码入站MES校验结果（步）
LD D1016.05  ; RK_02 电芯进料机构扫码触发（步）
ANDNOT P_On
ORLD
ANDLD
AND W65.02  ; RK_02 电芯进料机构扫码失败
ANDNOT C0050  ; 电芯进料机构扫码NG后重复次数计数
ANDNOT H8.00  ; 电芯进料机构重复扫码模式选择（0=使用/1=屏蔽）
UP(521)
OUT W65.05  ; RK_02 电芯进料机构重新扫码触发
LD W65.03  ; RK_02 电芯进料机构扫码成功
@OR H16.03  ; RK_02 电芯进料机构扫码完成记忆  // 可改为常开？
CNTX(546) 0050 D199  ; NG扫码重试次数设置, 电芯进料机构扫码NG后重复次数计数
; rung 11: 电芯进料机构步序跳转 / ********************************* / MES校验暂不参与到步序跳转程序
LD P_On
OUT TR0
AND D1013.00  ; RK_02 电芯进料机构单步/自动循环运行中（总）
AND D1016.06  ; RK_02 电芯进料机构扫码结果&扫码入站MES校验结果（步）
AND W65.02  ; RK_02 电芯进料机构扫码失败
AND W65.05  ; RK_02 电芯进料机构重新扫码触发
ANDNOT H8.00  ; 电芯进料机构重复扫码模式选择（0=使用/1=屏蔽）
RSET W65.00  ; RK_02 电芯进料机构扫码
@MOV(021) &32 D1016  ; RK_02 电芯进料机构步序  // RK_02 电芯进料机构扫码触发步（D1016.05）
LD TR0
%AND D1017.00  ; RK_02 电芯进料机构复位（M）
AND H15.00  ; RK_02 U0_Y 电芯进料X轴回原点记忆
AND 851.01  ; RK_02 U0_Y 电芯进料X轴取料位标志
AND H15.01  ; RK_02 U0_Z 电芯进料Z轴回原点记忆
AND 852.00  ; RK_02 U0_Z 电芯进料Z轴待料位（扫码）标志
AND H16.00  ; RK_02 电芯进料机构夹爪有料记忆
AND 800.00  ; RK_02 电芯进料机械手夹爪气缸夹紧位标志[0000.00]
AND 100.02  ; RK_02 电芯进料机械手压紧气缸伸出
OUT TR0
ANDNOT H16.03  ; RK_02 电芯进料机构扫码完成记忆
ANDNOT H16.04  ; RK_02 电芯进料机构夹爪有扫码OK料记忆
ANDNOT H16.05  ; RK_02 电芯进料机构夹爪有扫码NG料记忆
MOV(021) &16 D1016  ; RK_02 电芯进料机构步序  // RK_02 电芯进料机构进料Z轴待料位（扫码）&扫码数据初始化步（D1016.04）
LD TR0
AND H16.03  ; RK_02 电芯进料机构扫码完成记忆
LD H16.04  ; RK_02 电芯进料机构夹爪有扫码OK料记忆
OR H16.05  ; RK_02 电芯进料机构夹爪有扫码NG料记忆
ANDLD
MOV(021) &64 D1016  ; RK_02 电芯进料机构步序  // RK_02 电芯进料机构扫码&MES校验结果步（D1016.06）

